gfCNCPoint3[15642] = {X 203.9653, Y 32.4217, Z -4.6667, A 0.000, B 0.000, C 0.000 }
gfCNCPoint3[15643] = {X 206.9865, Y 38.6634, Z -4.6667, A 0.000, B 0.000, C 0.000 }
gfCNCPoint3[15644] = {X 207.4240, Y 39.8017, Z -4.6667, A 0.000, B 0.000, C 0.000 }
gfCNCPoint3[15645] = {X 207.6653, Y 40.9971, Z -4.6667, A 0.000, B 0.000, C 0.000 }
gfCNCPoint3[15646] = {X 207.7038, Y 42.2159, Z -4.6667, A 0.000, B 0.000, C 0.000 }
gfCNCPoint3[15647] = {X 207.5382, Y 43.4241, Z -4.6667, A 0.000, B 0.000, C 0.000 }
gfCNCPoint3[15648] = {X 207.1733, Y 44.5877, Z -4.6667, A 0.000, B 0.000, C 0.000 }
gfCNCPoint3[15649] = {X 206.6193, Y 45.6741, Z -4.6667, A 0.000, B 0.000, C 0.000 }
gfCNCPoint3[15650] = {X 205.8917, Y 46.6527, Z -4.6667, A 0.000, B 0.000, C 0.000 }
gfCNCPoint3[15651] = {X 205.0110, Y 47.4962, Z -4.6667, A 0.000, B 0.000, C 0.000 }
gfCNCPoint3[15652] = {X 204.4743, Y 47.9301, Z -4.6667, A 0.000, B 0.000, C 0.000 }
gfCNCPoint3[15653] = {X 203.5894, Y 48.5431, Z -4.6667, A 0.000, B 0.000, C 0.000 }
gfCNCPoint3[15654] = {X 202.6239, Y 49.0192, Z -4.6667, A 0.000, B 0.000, C 0.000 }
gfCNCPoint3[15655] = {X 201.4894, Y 49.3733, Z -4.6667, A 0.000, B 0.000, C 0.000 }
gfCNCPoint3[15656] = {X 200.3125, Y 49.5385, Z -4.6667, A 0.000, B 0.000, C 0.000 }
gfCNCPoint3[15657] = {X 199.1244, Y 49.5104, Z -4.6667, A 0.000, B 0.000, C 0.000 }
gfCNCPoint3[15658] = {X 196.8334, Y 50.6071, Z -4.6667, A 0.000, B 0.000, C 0.000 }
gfCNCPoint3[15659] = {X 194.4619, Y 51.5166, Z -4.6667, A 0.000, B 0.000, C 0.000 }
gfCNCPoint3[15660] = {X 192.0251, Y 52.2331, Z -4.6667, A 0.000, B 0.000, C 0.000 }
gfCNCPoint3[15661] = {X 190.7222, Y 52.5186, Z -4.6667, A 0.000, B 0.000, C 0.000 }
gfCNCPoint3[15662] = {X 189.4062, Y 52.7359, Z -4.6667, A 0.000, B 0.000, C 0.000 }
gfCNCPoint3[15663] = {X 189.9006, Y 53.9116, Z -4.6667, A 0.000, B 0.000, C 0.000 }
gfCNCPoint3[15664] = {X 190.2683, Y 55.1329, Z -4.6667, A 0.000, B 0.000, C 0.000 }
gfCNCPoint3[15665] = {X 190.5269, Y 56.5561, Z -4.6667, A 0.000, B 0.000, C 0.000 }
gfCNCPoint3[15666] = {X 190.6135, Y 58.0000, Z -4.6667, A 0.000, B 0.000, C 0.000 }
gfCNCPoint3[15667] = {X 190.6132, Y 58.8764, Z -4.6667, A 0.000, B 0.000, C 0.000 }
gfCNCPoint3[15668] = {X 208.6256, Y 78.5346, Z -4.6667, A 0.000, B 0.000, C 0.000 }
gfCNCPoint3[15669] = {X 206.8561, Y 80.1560, Z -4.6667, A 0.000, B 0.000, C 0.000 }
gfCNCPoint3[15670] = {X 213.5228, Y 87.4318, Z -4.6667, A 0.000, B 0.000, C 0.000 }
gfCNCPoint3[15671] = {X 214.2178, Y 87.3794, Z -4.6667, A 0.000, B 0.000, C 0.000 }
gfCNCPoint3[15672] = {X 214.9136, Y 87.3378, Z -4.6667, A 0.000, B 0.000, C 0.000 }
gfCNCPoint3[15673] = {X 234.0915, Y 75.0517, Z -4.6667, A 0.000, B 0.000, C 0.000 }
gfCNCPoint3[15674] = {X 219.6587, Y 69.3879, Z -4.6667, A 0.000, B 0.000, C 0.000 }
gfCNCPoint3[15675] = {X 218.4694, Y 68.9877, Z -4.6667, A 0.000, B 0.000, C 0.000 }
gfCNCPoint3[15676] = {X 217.2420, Y 68.7267, Z -4.6667, A 0.000, B 0.000, C 0.000 }
gfCNCPoint3[15677] = {X 215.9928, Y 68.6082, Z -4.6667, A 0.000, B 0.000, C 0.000 }
gfCNCPoint3[15678] = {X 214.5225, Y 68.4437, Z -4.6667, A 0.000, B 0.000, C 0.000 }
gfCNCPoint3[15679] = {X 213.0946, Y 68.0571, Z -4.6667, A 0.000, B 0.000, C 0.000 }
gfCNCPoint3[15680] = {X 211.7422, Y 67.4574, Z -4.6667, A 0.000, B 0.000, C 0.000 }
gfCNCPoint3[15681] = {X 210.4970, Y 66.6586, Z -4.6667, A 0.000, B 0.000, C 0.000 }
gfCNCPoint3[15682] = {X 209.3880, Y 65.6794, Z -4.6667, A 0.000, B 0.000, C 0.000 }
gfCNCPoint3[15683] = {X 208.4412, Y 64.5427, Z -4.6667, A 0.000, B 0.000, C 0.000 }
gfCNCPoint3[15684] = {X 207.6787, Y 63.2750, Z -4.6667, A 0.000, B 0.000, C 0.000 }
gfCNCPoint3[15685] = {X 207.1183, Y 61.9059, Z -4.6667, A 0.000, B 0.000, C 0.000 }
gfCNCPoint3[15686] = {X 206.7730, Y 60.4673, Z -4.6667, A 0.000, B 0.000, C 0.000 }
gfCNCPoint3[15687] = {X 206.6510, Y 58.9930, Z -4.6667, A 0.000, B 0.000, C 0.000 }
gfCNCPoint3[15688] = {X 206.6508, Y 58.0000, Z -4.6667, A 0.000, B 0.000, C 0.000 }
gfCNCPoint3[15689] = {X 206.7577, Y 56.5655, Z -4.6667, A 0.000, B 0.000, C 0.000 }
gfCNCPoint3[15690] = {X 207.0759, Y 55.1628, Z -4.6667, A 0.000, B 0.000, C 0.000 }
gfCNCPoint3[15691] = {X 207.5986, Y 53.8226, Z -4.6667, A 0.000, B 0.000, C 0.000 }
gfCNCPoint3[15692] = {X 208.3140, Y 52.5747, Z -4.6667, A 0.000, B 0.000, C 0.000 }
gfCNCPoint3[15693] = {X 209.2065, Y 51.4466, Z -4.6667, A 0.000, B 0.000, C 0.000 }
gfCNCPoint3[15694] = {X 210.2563, Y 50.4632, Z -4.6667, A 0.000, B 0.000, C 0.000 }
gfCNCPoint3[15695] = {X 211.4402, Y 49.6463, Z -4.6667, A 0.000, B 0.000, C 0.000 }
gfCNCPoint3[15696] = {X 212.5893, Y 49.0723, Z -4.6667, A 0.000, B 0.000, C 0.000 }
gfCNCPoint3[15697] = {X 213.8042, Y 48.6556, Z -4.6667, A 0.000, B 0.000, C 0.000 }
gfCNCPoint3[15698] = {X 213.2578, Y 48.0874, Z -4.6667, A 0.000, B 0.000, C 0.000 }
gfCNCPoint3[15699] = {X 212.8100, Y 47.4386, Z -4.6667, A 0.000, B 0.000, C 0.000 }
gfCNCPoint3[15700] = {X 212.4725, Y 46.7262, Z -4.6667, A 0.000, B 0.000, C 0.000 }
gfCNCPoint3[15701] = {X 212.2401, Y 45.8965, Z -4.6667, A 0.000, B 0.000, C 0.000 }
gfCNCPoint3[15702] = {X 212.1572, Y 45.0389, Z -4.6667, A 0.000, B 0.000, C 0.000 }
gfCNCPoint3[15703] = {X 212.1570, Y 44.1958, Z -4.6667, A 0.000, B 0.000, C 0.000 }
gfCNCPoint3[15704] = {X 212.2383, Y 43.3151, Z -4.6667, A 0.000, B 0.000, C 0.000 }
gfCNCPoint3[15705] = {X 212.4795, Y 42.4642, Z -4.6667, A 0.000, B 0.000, C 0.000 }
gfCNCPoint3[15706] = {X 212.8723, Y 41.6718, Z -4.6667, A 0.000, B 0.000, C 0.000 }
gfCNCPoint3[15707] = {X 213.4036, Y 40.9647, Z -4.6667, A 0.000, B 0.000, C 0.000 }
gfCNCPoint3[15708] = {X 213.6821, Y 40.6575, Z -4.6667, A 0.000, B 0.000, C 0.000 }
gfCNCPoint3[15709] = {X 213.6849, Y 40.3041, Z -4.6667, A 0.000, B 0.000, C 0.000 }
gfCNCPoint3[15710] = {X 213.6849, Y 17.4645, Z -4.6667, A 0.000, B 0.000, C 0.000 }
gfCNCPoint3[15711] = {X 213.6795, Y 16.7696, Z -4.6667, A 0.000, B 0.000, C 0.000 }
gfCNCPoint3[15712] = {X 213.6793, Y 16.5192, Z -4.6667, A 0.000, B 0.000, C 0.000 }
gfCNCPoint3[15713] = {X 213.0402, Y 15.7779, Z -4.6667, A 0.000, B 0.000, C 0.000 }
gfCNCPoint3[15714] = {X 212.5618, Y 14.9240, Z -4.6667, A 0.000, B 0.000, C 0.000 }
gfCNCPoint3[15715] = {X 212.2635, Y 13.9918, Z -4.6667, A 0.000, B 0.000, C 0.000 }
gfCNCPoint3[15716] = {X 212.1572, Y 13.0188, Z -4.6667, A 0.000, B 0.000, C 0.000 }
gfCNCPoint3[15717] = {X 212.1570, Y 12.1868, Z -4.6667, A 0.000, B 0.000, C 0.000 }
gfCNCPoint3[15718] = {X 212.2436, Y 11.2717, Z -4.6667, A 0.000, B 0.000, C 0.000 }
gfCNCPoint3[15719] = {X 212.5002, Y 10.3891, Z -4.6667, A 0.000, B 0.000, C 0.000 }
gfCNCPoint3[15720] = {X 212.9449, Y 9.5280, Z -4.6667, A 0.000, B 0.000, C 0.000 }
gfCNCPoint3[15721] = {X 213.5510, Y 8.7718, Z -4.6667, A 0.000, B 0.000, C 0.000 }
gfCNCPoint3[15722] = {X 214.2946, Y 8.1503, Z -4.6667, A 0.000, B 0.000, C 0.000 }
gfCNCPoint3[15723] = {X 215.1464, Y 7.6879, Z -4.6667, A 0.000, B 0.000, C 0.000 }
gfCNCPoint3[15724] = {X 216.0727, Y 7.4030, Z -4.6667, A 0.000, B 0.000, C 0.000 }
gfCNCPoint3[15725] = {X 217.0370, Y 7.3068, Z -4.6667, A 0.000, B 0.000, C 0.000 }
gfCNCPoint3[15726] = {X 223.4805, Y 7.3068, Z -4.6667, A 0.000, B 0.000, C 0.000 }
gfCNCPoint3[15727] = {X 224.4448, Y 7.4030, Z -4.6667, A 0.000, B 0.000, C 0.000 }
gfCNCPoint3[15728] = {X 225.3711, Y 7.6879, Z -4.6667, A 0.000, B 0.000, C 0.000 }
gfCNCPoint3[15729] = {X 226.2229, Y 8.1503, Z -4.6667, A 0.000, B 0.000, C 0.000 }
gfCNCPoint3[15730] = {X 226.9665, Y 8.7718, Z -4.6667, A 0.000, B 0.000, C 0.000 }
gfCNCPoint3[15731] = {X 227.5726, Y 9.5280, Z -4.6667, A 0.000, B 0.000, C 0.000 }
gfCNCPoint3[15732] = {X 228.0173, Y 10.3891, Z -4.6667, A 0.000, B 0.000, C 0.000 }
gfCNCPoint3[15733] = {X 228.2739, Y 11.2717, Z -4.6667, A 0.000, B 0.000, C 0.000 }
gfCNCPoint3[15734] = {X 228.3605, Y 12.1868, Z -4.6667, A 0.000, B 0.000, C 0.000 }
gfCNCPoint3[15735] = {X 228.3603, Y 13.0237, Z -4.6667, A 0.000, B 0.000, C 0.000 }
gfCNCPoint3[15736] = {X 228.2529, Y 13.9971, Z -4.6667, A 0.000, B 0.000, C 0.000 }
gfCNCPoint3[15737] = {X 227.9533, Y 14.9294, Z -4.6667, A 0.000, B 0.000, C 0.000 }
gfCNCPoint3[15738] = {X 227.4737, Y 15.7831, Z -4.6667, A 0.000, B 0.000, C 0.000 }
gfCNCPoint3[15739] = {X 226.8333, Y 16.5239, Z -4.6667, A 0.000, B 0.000, C 0.000 }
gfCNCPoint3[15740] = {X 226.8342, Y 40.6638, Z -4.6667, A 0.000, B 0.000, C 0.000 }
gfCNCPoint3[15741] = {X 227.4743, Y 41.4046, Z -4.6667, A 0.000, B 0.000, C 0.000 }
gfCNCPoint3[15742] = {X 227.9537, Y 42.2583, Z -4.6667, A 0.000, B 0.000, C 0.000 }
gfCNCPoint3[15743] = {X 228.2531, Y 43.1906, Z -4.6667, A 0.000, B 0.000, C 0.000 }
gfCNCPoint3[15744] = {X 228.3603, Y 44.1638, Z -4.6667, A 0.000, B 0.000, C 0.000 }
gfCNCPoint3[15745] = {X 228.3605, Y 45.0000, Z -4.6667, A 0.000, B 0.000, C 0.000 }
gfCNCPoint3[15746] = {X 228.3507, Y 45.3090, Z -4.6667, A 0.000, B 0.000, C 0.000 }
gfCNCPoint3[15747] = {X 228.3214, Y 45.6167, Z -4.6667, A 0.000, B 0.000, C 0.000 }
gfCNCPoint3[15748] = {X 228.0910, Y 46.5992, Z -4.6667, A 0.000, B 0.000, C 0.000 }
gfCNCPoint3[15749] = {X 227.6635, Y 47.5134, Z -4.6667, A 0.000, B 0.000, C 0.000 }
gfCNCPoint3[15750] = {X 227.0571, Y 48.3200, Z -4.6667, A 0.000, B 0.000, C 0.000 }
gfCNCPoint3[15751] = {X 226.7053, Y 47.9934, Z -4.6667, A 0.000, B 0.000, C 0.000 }
gfCNCPoint3[15752] = {X 226.0261, Y 48.5889, Z -4.6667, A 0.000, B 0.000, C 0.000 }
gfCNCPoint3[15753] = {X 225.2396, Y 49.0331, Z -4.6667, A 0.000, B 0.000, C 0.000 }
gfCNCPoint3[15754] = {X 224.3790, Y 49.3073, Z -4.6667, A 0.000, B 0.000, C 0.000 }
gfCNCPoint3[15755] = {X 223.4805, Y 49.4000, Z -4.6667, A 0.000, B 0.000, C 0.000 }
gfCNCPoint3[15756] = {X 217.0370, Y 49.4000, Z -4.6667, A 0.000, B 0.000, C 0.000 }
gfCNCPoint3[15757] = {X 216.0579, Y 49.2897, Z -4.6667, A 0.000, B 0.000, C 0.000 }
gfCNCPoint3[15758] = {X 215.1279, Y 48.9643, Z -4.6667, A 0.000, B 0.000, C 0.000 }
gfCNCPoint3[15759] = {X 214.2936, Y 48.4400, Z -4.6667, A 0.000, B 0.000, C 0.000 }
gfCNCPoint3[15760] = {X 213.5969, Y 47.7433, Z -4.6667, A 0.000, B 0.000, C 0.000 }
gfCNCPoint3[15761] = {X 213.0727, Y 46.9091, Z -4.6667, A 0.000, B 0.000, C 0.000 }
gfCNCPoint3[15762] = {X 212.7473, Y 45.9791, Z -4.6667, A 0.000, B 0.000, C 0.000 }
gfCNCPoint3[15763] = {X 212.6370, Y 45.0000, Z -4.6667, A 0.000, B 0.000, C 0.000 }
gfCNCPoint3[15764] = {X 212.6370, Y 44.1958, Z -4.6667, A 0.000, B 0.000, C 0.000 }
gfCNCPoint3[15765] = {X 212.7102, Y 43.4029, Z -4.6667, A 0.000, B 0.000, C 0.000 }
gfCNCPoint3[15766] = {X 212.9273, Y 42.6369, Z -4.6667, A 0.000, B 0.000, C 0.000 }
gfCNCPoint3[15767] = {X 213.2810, Y 41.9236, Z -4.6667, A 0.000, B 0.000, C 0.000 }
gfCNCPoint3[15768] = {X 213.7592, Y 41.2871, Z -4.6667, A 0.000, B 0.000, C 0.000 }
gfCNCPoint3[15769] = {X 214.1607, Y 40.8442, Z -4.6667, A 0.000, B 0.000, C 0.000 }
gfCNCPoint3[15770] = {X 214.1649, Y 40.3060, Z -4.6667, A 0.000, B 0.000, C 0.000 }
gfCNCPoint3[15771] = {X 214.1649, Y 17.4626, Z -4.6667, A 0.000, B 0.000, C 0.000 }
gfCNCPoint3[15772] = {X 214.1595, Y 16.7692, Z -4.6667, A 0.000, B 0.000, C 0.000 }
gfCNCPoint3[15773] = {X 214.1591, Y 16.3063, Z -4.6667, A 0.000, B 0.000, C 0.000 }
gfCNCPoint3[15774] = {X 213.5167, Y 15.6176, Z -4.6667, A 0.000, B 0.000, C 0.000 }
gfCNCPoint3[15775] = {X 213.0356, Y 14.8079, Z -4.6667, A 0.000, B 0.000, C 0.000 }
gfCNCPoint3[15776] = {X 212.7378, Y 13.9144, Z -4.6667, A 0.000, B 0.000, C 0.000 }
gfCNCPoint3[15777] = {X 212.6370, Y 12.9779, Z -4.6667, A 0.000, B 0.000, C 0.000 }
gfCNCPoint3[15778] = {X 212.6370, Y 12.1868, Z -4.6667, A 0.000, B 0.000, C 0.000 }
gfCNCPoint3[15779] = {X 212.7473, Y 11.2077, Z -4.6667, A 0.000, B 0.000, C 0.000 }
gfCNCPoint3[15780] = {X 213.0728, Y 10.2777, Z -4.6667, A 0.000, B 0.000, C 0.000 }
gfCNCPoint3[15781] = {X 213.5970, Y 9.4435, Z -4.6667, A 0.000, B 0.000, C 0.000 }
gfCNCPoint3[15782] = {X 214.2937, Y 8.7468, Z -4.6667, A 0.000, B 0.000, C 0.000 }
gfCNCPoint3[15783] = {X 215.1279, Y 8.2226, Z -4.6667, A 0.000, B 0.000, C 0.000 }
gfCNCPoint3[15784] = {X 216.0579, Y 7.8971, Z -4.6667, A 0.000, B 0.000, C 0.000 }
gfCNCPoint3[15785] = {X 217.0370, Y 7.7868, Z -4.6667, A 0.000, B 0.000, C 0.000 }
gfCNCPoint3[15786] = {X 223.4805, Y 7.7868, Z -4.6667, A 0.000, B 0.000, C 0.000 }
gfCNCPoint3[15787] = {X 224.4596, Y 7.8971, Z -4.6667, A 0.000, B 0.000, C 0.000 }
gfCNCPoint3[15788] = {X 225.3896, Y 8.2226, Z -4.6667, A 0.000, B 0.000, C 0.000 }
gfCNCPoint3[15789] = {X 226.2238, Y 8.7468, Z -4.6667, A 0.000, B 0.000, C 0.000 }
gfCNCPoint3[15790] = {X 226.9205, Y 9.4435, Z -4.6667, A 0.000, B 0.000, C 0.000 }
gfCNCPoint3[15791] = {X 227.4447, Y 10.2777, Z -4.6667, A 0.000, B 0.000, C 0.000 }
gfCNCPoint3[15792] = {X 227.7702, Y 11.2077, Z -4.6667, A 0.000, B 0.000, C 0.000 }
gfCNCPoint3[15793] = {X 227.8805, Y 12.1868, Z -4.6667, A 0.000, B 0.000, C 0.000 }
gfCNCPoint3[15794] = {X 227.8802, Y 13.0233, Z -4.6667, A 0.000, B 0.000, C 0.000 }
gfCNCPoint3[15795] = {X 227.7720, Y 13.9493, Z -4.6667, A 0.000, B 0.000, C 0.000 }
gfCNCPoint3[15796] = {X 227.4710, Y 14.8316, Z -4.6667, A 0.000, B 0.000, C 0.000 }
gfCNCPoint3[15797] = {X 226.9909, Y 15.6307, Z -4.6667, A 0.000, B 0.000, C 0.000 }
gfCNCPoint3[15798] = {X 226.3532, Y 16.3108, Z -4.6667, A 0.000, B 0.000, C 0.000 }
gfCNCPoint3[15799] = {X 226.3542, Y 40.8768, Z -4.6667, A 0.000, B 0.000, C 0.000 }
gfCNCPoint3[15800] = {X 226.9983, Y 41.5659, Z -4.6667, A 0.000, B 0.000, C 0.000 }
gfCNCPoint3[15801] = {X 227.4808, Y 42.3764, Z -4.6667, A 0.000, B 0.000, C 0.000 }
gfCNCPoint3[15802] = {X 227.7794, Y 43.2711, Z -4.6667, A 0.000, B 0.000, C 0.000 }
gfCNCPoint3[15803] = {X 227.8805, Y 44.2089, Z -4.6667, A 0.000, B 0.000, C 0.000 }
gfCNCPoint3[15804] = {X 227.8805, Y 45.0000, Z -4.6667, A 0.000, B 0.000, C 0.000 }
gfCNCPoint3[15805] = {X 227.8037, Y 45.8182, Z -4.6667, A 0.000, B 0.000, C 0.000 }
gfCNCPoint3[15806] = {X 227.5762, Y 46.6079, Z -4.6667, A 0.000, B 0.000, C 0.000 }
gfCNCPoint3[15807] = {X 227.2057, Y 47.3415, Z -4.6667, A 0.000, B 0.000, C 0.000 }
gfCNCPoint3[15808] = {X 226.7053, Y 47.9934, Z -4.6667, A 0.000, B 0.000, C 0.000 }
gfCNCPoint3[15809] = {X 227.0571, Y 48.3200, Z -4.6667, A 0.000, B 0.000, C 0.000 }
gfCNCPoint3[15810] = {X 236.2309, Y 48.3200, Z -4.6667, A 0.000, B 0.000, C 0.000 }
gfCNCPoint3[15811] = {X 235.6245, Y 47.5134, Z -4.6667, A 0.000, B 0.000, C 0.000 }
gfCNCPoint3[15812] = {X 235.1970, Y 46.5992, Z -4.6667, A 0.000, B 0.000, C 0.000 }
gfCNCPoint3[15813] = {X 234.9666, Y 45.6167, Z -4.6667, A 0.000, B 0.000, C 0.000 }
gfCNCPoint3[15814] = {X 234.9373, Y 45.3090, Z -4.6667, A 0.000, B 0.000, C 0.000 }
gfCNCPoint3[15815] = {X 234.9275, Y 45.0000, Z -4.6667, A 0.000, B 0.000, C 0.000 }
gfCNCPoint3[15816] = {X 234.9275, Y 44.2089, Z -4.6667, A 0.000, B 0.000, C 0.000 }
gfCNCPoint3[15817] = {X 235.0194, Y 43.2661, Z -4.6667, A 0.000, B 0.000, C 0.000 }
gfCNCPoint3[15818] = {X 235.2917, Y 42.3588, Z -4.6667, A 0.000, B 0.000, C 0.000 }
gfCNCPoint3[15819] = {X 235.7342, Y 41.5212, Z -4.6667, A 0.000, B 0.000, C 0.000 }
gfCNCPoint3[15820] = {X 236.3302, Y 40.7849, Z -4.6667, A 0.000, B 0.000, C 0.000 }
gfCNCPoint3[15821] = {X 237.0572, Y 40.1776, Z -4.6667, A 0.000, B 0.000, C 0.000 }
gfCNCPoint3[15822] = {X 237.8878, Y 39.7222, Z -4.6667, A 0.000, B 0.000, C 0.000 }
gfCNCPoint3[15823] = {X 241.5463, Y 32.5611, Z -4.6667, A 0.000, B 0.000, C 0.000 }
gfCNCPoint3[15824] = {X 240.2118, Y 31.5584, Z -4.6667, A 0.000, B 0.000, C 0.000 }
gfCNCPoint3[15825] = {X 239.0310, Y 30.3785, Z -4.6667, A 0.000, B 0.000, C 0.000 }
gfCNCPoint3[15826] = {X 238.0273, Y 29.0447, Z -4.6667, A 0.000, B 0.000, C 0.000 }
gfCNCPoint3[15827] = {X 237.2205, Y 27.5834, Z -4.6667, A 0.000, B 0.000, C 0.000 }
gfCNCPoint3[15828] = {X 236.6265, Y 26.0235, Z -4.6667, A 0.000, B 0.000, C 0.000 }
gfCNCPoint3[15829] = {X 236.1914, Y 24.1499, Z -4.6667, A 0.000, B 0.000, C 0.000 }
gfCNCPoint3[15830] = {X 235.9695, Y 22.2393, Z -4.6667, A 0.000, B 0.000, C 0.000 }
gfCNCPoint3[15831] = {X 235.9636, Y 20.3158, Z -4.6667, A 0.000, B 0.000, C 0.000 }
gfCNCPoint3[15832] = {X 236.1739, Y 18.4039, Z -4.6667, A 0.000, B 0.000, C 0.000 }
gfCNCPoint3[15833] = {X 236.5975, Y 16.5277, Z -4.6667, A 0.000, B 0.000, C 0.000 }
gfCNCPoint3[15834] = {X 237.1169, Y 15.0571, Z -4.6667, A 0.000, B 0.000, C 0.000 }
gfCNCPoint3[15835] = {X 237.8166, Y 13.6632, Z -4.6667, A 0.000, B 0.000, C 0.000 }
gfCNCPoint3[15836] = {X 238.6856, Y 12.3681, Z -4.6667, A 0.000, B 0.000, C 0.000 }
gfCNCPoint3[15837] = {X 239.7103, Y 11.1923, Z -4.6667, A 0.000, B 0.000, C 0.000 }
gfCNCPoint3[15838] = {X 240.8746, Y 10.1541, Z -4.6667, A 0.000, B 0.000, C 0.000 }
gfCNCPoint3[15839] = {X 242.1599, Y 9.2702, Z -4.6667, A 0.000, B 0.000, C 0.000 }
gfCNCPoint3[15840] = {X 243.5460, Y 8.5546, Z -4.6667, A 0.000, B 0.000, C 0.000 }
gfCNCPoint3[15841] = {X 245.0110, Y 8.0185, Z -4.6667, A 0.000, B 0.000, C 0.000 }
gfCNCPoint3[15842] = {X 246.5316, Y 7.6705, Z -4.6667, A 0.000, B 0.000, C 0.000 }
gfCNCPoint3[15843] = {X 248.6761, Y 7.3930, Z -4.6667, A 0.000, B 0.000, C 0.000 }
gfCNCPoint3[15844] = {X 250.8369, Y 7.3106, Z -4.6667, A 0.000, B 0.000, C 0.000 }
gfCNCPoint3[15845] = {X 266.7608, Y 7.3106, Z -4.6667, A 0.000, B 0.000, C 0.000 }
gfCNCPoint3[15846] = {X 267.7191, Y 7.4120, Z -4.6667, A 0.000, B 0.000, C 0.000 }
gfCNCPoint3[15847] = {X 268.6388, Y 7.6997, Z -4.6667, A 0.000, B 0.000, C 0.000 }
gfCNCPoint3[15848] = {X 269.4841, Y 8.1624, Z -4.6667, A 0.000, B 0.000, C 0.000 }
gfCNCPoint3[15849] = {X 270.2221, Y 8.7821, Z -4.6667, A 0.000, B 0.000, C 0.000 }
gfCNCPoint3[15850] = {X 270.8239, Y 9.5347, Z -4.6667, A 0.000, B 0.000, C 0.000 }
gfCNCPoint3[15851] = {X 271.2663, Y 10.3908, Z -4.6667, A 0.000, B 0.000, C 0.000 }
gfCNCPoint3[15852] = {X 271.5234, Y 11.2719, Z -4.6667, A 0.000, B 0.000, C 0.000 }
gfCNCPoint3[15853] = {X 271.6110, Y 12.1855, Z -4.6667, A 0.000, B 0.000, C 0.000 }
gfCNCPoint3[15854] = {X 271.6108, Y 13.0237, Z -4.6667, A 0.000, B 0.000, C 0.000 }
gfCNCPoint3[15855] = {X 271.5128, Y 13.9524, Z -4.6667, A 0.000, B 0.000, C 0.000 }
gfCNCPoint3[15856] = {X 271.2396, Y 14.8453, Z -4.6667, A 0.000, B 0.000, C 0.000 }
gfCNCPoint3[15857] = {X 275.6743, Y 16.6820, Z -4.6667, A 0.000, B 0.000, C 0.000 }
gfCNCPoint3[15858] = {X 275.3127, Y 17.4566, Z -4.6667, A 0.000, B 0.000, C 0.000 }
gfCNCPoint3[15859] = {X 274.8840, Y 18.1964, Z -4.6667, A 0.000, B 0.000, C 0.000 }
gfCNCPoint3[15860] = {X 274.8839, Y 38.9902, Z -4.6667, A 0.000, B 0.000, C 0.000 }
gfCNCPoint3[15861] = {X 275.3140, Y 39.7327, Z -4.6667, A 0.000, B 0.000, C 0.000 }
gfCNCPoint3[15862] = {X 275.6766, Y 40.5104, Z -4.6667, A 0.000, B 0.000, C 0.000 }
gfCNCPoint3[15863] = {X 276.0377, Y 39.7359, Z -4.6667, A 0.000, B 0.000, C 0.000 }
gfCNCPoint3[15864] = {X 276.4653, Y 38.9961, Z -4.6667, A 0.000, B 0.000, C 0.000 }
gfCNCPoint3[15865] = {X 276.4649, Y 18.1968, Z -4.6667, A 0.000, B 0.000, C 0.000 }
gfCNCPoint3[15866] = {X 276.0362, Y 17.4569, Z -4.6667, A 0.000, B 0.000, C 0.000 }
gfCNCPoint3[15867] = {X 275.6743, Y 16.6820, Z -4.6667, A 0.000, B 0.000, C 0.000 }
gfCNCPoint3[15868] = {X 273.4570, Y 15.7637, Z -4.6667, A 0.000, B 0.000, C 0.000 }
gfCNCPoint3[15869] = {X 273.0265, Y 16.6339, Z -4.6667, A 0.000, B 0.000, C 0.000 }
gfCNCPoint3[15870] = {X 272.4840, Y 17.4391, Z -4.6667, A 0.000, B 0.000, C 0.000 }
gfCNCPoint3[15871] = {X 272.4839, Y 39.7475, Z -4.6667, A 0.000, B 0.000, C 0.000 }
gfCNCPoint3[15872] = {X 273.0276, Y 40.5547, Z -4.6667, A 0.000, B 0.000, C 0.000 }
gfCNCPoint3[15873] = {X 273.4587, Y 41.4273, Z -4.6667, A 0.000, B 0.000, C 0.000 }
gfCNCPoint3[15874] = {X 273.7589, Y 42.3094, Z -4.6667, A 0.000, B 0.000, C 0.000 }
gfCNCPoint3[15875] = {X 273.9439, Y 43.2225, Z -4.6667, A 0.000, B 0.000, C 0.000 }
gfCNCPoint3[15876] = {X 274.0108, Y 44.1519, Z -4.6667, A 0.000, B 0.000, C 0.000 }
gfCNCPoint3[15877] = {X 274.0110, Y 45.0000, Z -4.6667, A 0.000, B 0.000, C 0.000 }
gfCNCPoint3[15878] = {X 273.9884, Y 45.5734, Z -4.6667, A 0.000, B 0.000, C 0.000 }
gfCNCPoint3[15879] = {X 273.9207, Y 46.1433, Z -4.6667, A 0.000, B 0.000, C 0.000 }
gfCNCPoint3[15880] = {X 275.0713, Y 45.9760, Z -4.6667, A 0.000, B 0.000, C 0.000 }
gfCNCPoint3[15881] = {X 276.2327, Y 45.9200, Z -4.6667, A 0.000, B 0.000, C 0.000 }
gfCNCPoint3[15882] = {X 277.3960, Y 45.9200, Z -4.6667, A 0.000, B 0.000, C 0.000 }
gfCNCPoint3[15883] = {X 277.3539, Y 45.4857, Z -4.6667, A 0.000, B 0.000, C 0.000 }
gfCNCPoint3[15884] = {X 277.3378, Y 45.0498, Z -4.6667, A 0.000, B 0.000, C 0.000 }
gfCNCPoint3[15885] = {X 277.3377, Y 44.1984, Z -4.6667, A 0.000, B 0.000, C 0.000 }
gfCNCPoint3[15886] = {X 277.4029, Y 43.2534, Z -4.6667, A 0.000, B 0.000, C 0.000 }
gfCNCPoint3[15887] = {X 277.5895, Y 42.3247, Z -4.6667, A 0.000, B 0.000, C 0.000 }
gfCNCPoint3[15888] = {X 277.8943, Y 41.4279, Z -4.6667, A 0.000, B 0.000, C 0.000 }
gfCNCPoint3[15889] = {X 278.3242, Y 40.5572, Z -4.6667, A 0.000, B 0.000, C 0.000 }
gfCNCPoint3[15890] = {X 278.8653, Y 39.7510, Z -4.6667, A 0.000, B 0.000, C 0.000 }
gfCNCPoint3[15891] = {X 278.8649, Y 17.4394, Z -4.6667, A 0.000, B 0.000, C 0.000 }
gfCNCPoint3[15892] = {X 278.3223, Y 16.6341, Z -4.6667, A 0.000, B 0.000, C 0.000 }
gfCNCPoint3[15893] = {X 277.8917, Y 15.7637, Z -4.6667, A 0.000, B 0.000, C 0.000 }
gfCNCPoint3[15894] = {X 277.5902, Y 14.8788, Z -4.6667, A 0.000, B 0.000, C 0.000 }
gfCNCPoint3[15895] = {X 277.4046, Y 13.9627, Z -4.6667, A 0.000, B 0.000, C 0.000 }
gfCNCPoint3[15896] = {X 277.3379, Y 13.0303, Z -4.6667, A 0.000, B 0.000, C 0.000 }
gfCNCPoint3[15897] = {X 277.3377, Y 12.1868, Z -4.6667, A 0.000, B 0.000, C 0.000 }
gfCNCPoint3[15898] = {X 277.3952, Y 11.2737, Z -4.6667, A 0.000, B 0.000, C 0.000 }
gfCNCPoint3[15899] = {X 277.5667, Y 10.3750, Z -4.6667, A 0.000, B 0.000, C 0.000 }
gfCNCPoint3[15900] = {X 277.8496, Y 9.5050, Z -4.6667, A 0.000, B 0.000, C 0.000 }
gfCNCPoint3[15901] = {X 273.4968, Y 9.5050, Z -4.6667, A 0.000, B 0.000, C 0.000 }
gfCNCPoint3[15902] = {X 273.7800, Y 10.3733, Z -4.6667, A 0.000, B 0.000, C 0.000 }
gfCNCPoint3[15903] = {X 273.9524, Y 11.2703, Z -4.6667, A 0.000, B 0.000, C 0.000 }
gfCNCPoint3[15904] = {X 274.0110, Y 12.1819, Z -4.6667, A 0.000, B 0.000, C 0.000 }
gfCNCPoint3[15905] = {X 274.0107, Y 13.0462, Z -4.6667, A 0.000, B 0.000, C 0.000 }
gfCNCPoint3[15906] = {X 273.9427, Y 13.9732, Z -4.6667, A 0.000, B 0.000, C 0.000 }
gfCNCPoint3[15907] = {X 273.7571, Y 14.8840, Z -4.6667, A 0.000, B 0.000, C 0.000 }
gfCNCPoint3[15908] = {X 273.4570, Y 15.7637, Z -4.6667, A 0.000, B 0.000, C 0.000 }
gfCNCPoint3[15909] = {X 271.2396, Y 14.8453, Z -4.6667, A 0.000, B 0.000, C 0.000 }
gfCNCPoint3[15910] = {X 270.7504, Y 15.7455, Z -4.6667, A 0.000, B 0.000, C 0.000 }
gfCNCPoint3[15911] = {X 270.0840, Y 16.5237, Z -4.6667, A 0.000, B 0.000, C 0.000 }
gfCNCPoint3[15912] = {X 270.0839, Y 40.6630, Z -4.6667, A 0.000, B 0.000, C 0.000 }
gfCNCPoint3[15913] = {X 270.7243, Y 41.4038, Z -4.6667, A 0.000, B 0.000, C 0.000 }
gfCNCPoint3[15914] = {X 271.2040, Y 42.2576, Z -4.6667, A 0.000, B 0.000, C 0.000 }
gfCNCPoint3[15915] = {X 271.5035, Y 43.1899, Z -4.6667, A 0.000, B 0.000, C 0.000 }
gfCNCPoint3[15916] = {X 271.6108, Y 44.1633, Z -4.6667, A 0.000, B 0.000, C 0.000 }
gfCNCPoint3[15917] = {X 271.6110, Y 45.0000, Z -4.6667, A 0.000, B 0.000, C 0.000 }
gfCNCPoint3[15918] = {X 271.5959, Y 45.3844, Z -4.6667, A 0.000, B 0.000, C 0.000 }
gfCNCPoint3[15919] = {X 271.5505, Y 45.7664, Z -4.6667, A 0.000, B 0.000, C 0.000 }
gfCNCPoint3[15920] = {X 271.2989, Y 46.7171, Z -4.6667, A 0.000, B 0.000, C 0.000 }
gfCNCPoint3[15921] = {X 270.8619, Y 47.5982, Z -4.6667, A 0.000, B 0.000, C 0.000 }
gfCNCPoint3[15922] = {X 270.2571, Y 48.3736, Z -4.6667, A 0.000, B 0.000, C 0.000 }
gfCNCPoint3[15923] = {X 269.5090, Y 49.0121, Z -4.6667, A 0.000, B 0.000, C 0.000 }
gfCNCPoint3[15924] = {X 268.6482, Y 49.4876, Z -4.6667, A 0.000, B 0.000, C 0.000 }
gfCNCPoint3[15925] = {X 267.7095, Y 49.7809, Z -4.6667, A 0.000, B 0.000, C 0.000 }
gfCNCPoint3[15926] = {X 266.7310, Y 49.8800, Z -4.6667, A 0.000, B 0.000, C 0.000 }
gfCNCPoint3[15927] = {X 262.1384, Y 49.8800, Z -4.6667, A 0.000, B 0.000, C 0.000 }
gfCNCPoint3[15928] = {X 262.1384, Y 54.6800, Z -4.6667, A 0.000, B 0.000, C 0.000 }
gfCNCPoint3[15929] = {X 260.2870, Y 54.6800, Z -4.6667, A 0.000, B 0.000, C 0.000 }
gfCNCPoint3[15930] = {X 261.9957, Y 55.3582, Z -4.6667, A 0.000, B 0.000, C 0.000 }
gfCNCPoint3[15931] = {X 262.0630, Y 55.0183, Z -4.6667, A 0.000, B 0.000, C 0.000 }
gfCNCPoint3[15932] = {X 262.1384, Y 54.6800, Z -4.6667, A 0.000, B 0.000, C 0.000 }
gfCNCPoint3[15933] = {X 262.1384, Y 52.2800, Z -4.6667, A 0.000, B 0.000, C 0.000 }
gfCNCPoint3[15934] = {X 260.2876, Y 52.2800, Z -4.6667, A 0.000, B 0.000, C 0.000 }
gfCNCPoint3[15935] = {X 259.1915, Y 52.1970, Z -4.6667, A 0.000, B 0.000, C 0.000 }
gfCNCPoint3[15936] = {X 258.1205, Y 51.9500, Z -4.6667, A 0.000, B 0.000, C 0.000 }
gfCNCPoint3[15937] = {X 257.0989, Y 51.5445, Z -4.6667, A 0.000, B 0.000, C 0.000 }
gfCNCPoint3[15938] = {X 256.1499, Y 50.9898, Z -4.6667, A 0.000, B 0.000, C 0.000 }
gfCNCPoint3[15939] = {X 255.2953, Y 50.2986, Z -4.6667, A 0.000, B 0.000, C 0.000 }
gfCNCPoint3[15940] = {X 253.6495, Y 52.0454, Z -4.6667, A 0.000, B 0.000, C 0.000 }
gfCNCPoint3[15941] = {X 253.4933, Y 51.8950, Z -4.6667, A 0.000, B 0.000, C 0.000 }
gfCNCPoint3[15942] = {X 253.3406, Y 51.7410, Z -4.6667, A 0.000, B 0.000, C 0.000 }
gfCNCPoint3[15943] = {X 253.2763, Y 51.8066, Z -4.6667, A 0.000, B 0.000, C 0.000 }
gfCNCPoint3[15944] = {X 253.2115, Y 51.8716, Z -4.6667, A 0.000, B 0.000, C 0.000 }
gfCNCPoint3[15945] = {X 253.6495, Y 52.0454, Z -4.6667, A 0.000, B 0.000, C 0.000 }
gfCNCPoint3[15946] = {X 255.2953, Y 50.2986, Z -4.6667, A 0.000, B 0.000, C 0.000 }
gfCNCPoint3[15947] = {X 255.1778, Y 50.1855, Z -4.6667, A 0.000, B 0.000, C 0.000 }
gfCNCPoint3[15948] = {X 255.0630, Y 50.0697, Z -4.6667, A 0.000, B 0.000, C 0.000 }
gfCNCPoint3[15949] = {X 254.3405, Y 49.1989, Z -4.6667, A 0.000, B 0.000, C 0.000 }
gfCNCPoint3[15950] = {X 253.7617, Y 48.2267, Z -4.6667, A 0.000, B 0.000, C 0.000 }
gfCNCPoint3[15951] = {X 253.3406, Y 47.1766, Z -4.6667, A 0.000, B 0.000, C 0.000 }
gfCNCPoint3[15952] = {X 252.9194, Y 48.2267, Z -4.6667, A 0.000, B 0.000, C 0.000 }
gfCNCPoint3[15953] = {X 252.3406, Y 49.1989, Z -4.6667, A 0.000, B 0.000, C 0.000 }
gfCNCPoint3[15954] = {X 251.6182, Y 50.0697, Z -4.6667, A 0.000, B 0.000, C 0.000 }
gfCNCPoint3[15955] = {X 251.5699, Y 50.1190, Z -4.6667, A 0.000, B 0.000, C 0.000 }
gfCNCPoint3[15956] = {X 251.5211, Y 50.1679, Z -4.6667, A 0.000, B 0.000, C 0.000 }
gfCNCPoint3[15957] = {X 250.7151, Y 50.8585, Z -4.6667, A 0.000, B 0.000, C 0.000 }
gfCNCPoint3[15958] = {X 249.8174, Y 51.4246, Z -4.6667, A 0.000, B 0.000, C 0.000 }
gfCNCPoint3[15959] = {X 248.8468, Y 51.8542, Z -4.6667, A 0.000, B 0.000, C 0.000 }
gfCNCPoint3[15960] = {X 247.8241, Y 52.1381, Z -4.6667, A 0.000, B 0.000, C 0.000 }
gfCNCPoint3[15961] = {X 247.8929, Y 52.2638, Z -4.6667, A 0.000, B 0.000, C 0.000 }
gfCNCPoint3[15962] = {X 247.9602, Y 52.3904, Z -4.6667, A 0.000, B 0.000, C 0.000 }
gfCNCPoint3[15963] = {X 250.9674, Y 53.5630, Z -4.6667, A 0.000, B 0.000, C 0.000 }
gfCNCPoint3[15964] = {X 264.1528, Y 58.7966, Z -4.6667, A 0.000, B 0.000, C 0.000 }
gfCNCPoint3[15965] = {X 264.1527, Y 58.0000, Z -4.6667, A 0.000, B 0.000, C 0.000 }
gfCNCPoint3[15966] = {X 264.2035, Y 56.8934, Z -4.6667, A 0.000, B 0.000, C 0.000 }
gfCNCPoint3[15967] = {X 264.3554, Y 55.7961, Z -4.6667, A 0.000, B 0.000, C 0.000 }
gfCNCPoint3[15968] = {X 264.4116, Y 55.5125, Z -4.6667, A 0.000, B 0.000, C 0.000 }
gfCNCPoint3[15969] = {X 264.4745, Y 55.2303, Z -4.6667, A 0.000, B 0.000, C 0.000 }
gfCNCPoint3[15970] = {X 264.9369, Y 53.7185, Z -4.6667, A 0.000, B 0.000, C 0.000 }
gfCNCPoint3[15971] = {X 265.5928, Y 52.2800, Z -4.6667, A 0.000, B 0.000, C 0.000 }
gfCNCPoint3[15972] = {X 262.1384, Y 52.2800, Z -4.6667, A 0.000, B 0.000, C 0.000 }
gfCNCPoint3[15973] = {X 262.1384, Y 49.8800, Z -4.6667, A 0.000, B 0.000, C 0.000 }
gfCNCPoint3[15974] = {X 260.2876, Y 49.8800, Z -4.6667, A 0.000, B 0.000, C 0.000 }
gfCNCPoint3[15975] = {X 259.2646, Y 49.7716, Z -4.6667, A 0.000, B 0.000, C 0.000 }
gfCNCPoint3[15976] = {X 258.2870, Y 49.4511, Z -4.6667, A 0.000, B 0.000, C 0.000 }
gfCNCPoint3[15977] = {X 257.3984, Y 48.9328, Z -4.6667, A 0.000, B 0.000, C 0.000 }
gfCNCPoint3[15978] = {X 256.6382, Y 48.2398, Z -4.6667, A 0.000, B 0.000, C 0.000 }
gfCNCPoint3[15979] = {X 256.0401, Y 47.4028, Z -4.6667, A 0.000, B 0.000, C 0.000 }
gfCNCPoint3[15980] = {X 255.6308, Y 46.4590, Z -4.6667, A 0.000, B 0.000, C 0.000 }
gfCNCPoint3[15981] = {X 255.4666, Y 45.7568, Z -4.6667, A 0.000, B 0.000, C 0.000 }
gfCNCPoint3[15982] = {X 255.4077, Y 45.0380, Z -4.6667, A 0.000, B 0.000, C 0.000 }
gfCNCPoint3[15983] = {X 255.4080, Y 44.1417, Z -4.6667, A 0.000, B 0.000, C 0.000 }
gfCNCPoint3[15984] = {X 255.5183, Y 43.1751, Z -4.6667, A 0.000, B 0.000, C 0.000 }
gfCNCPoint3[15985] = {X 255.8181, Y 42.2497, Z -4.6667, A 0.000, B 0.000, C 0.000 }
gfCNCPoint3[15986] = {X 256.2955, Y 41.4021, Z -4.6667, A 0.000, B 0.000, C 0.000 }
gfCNCPoint3[15987] = {X 256.9315, Y 40.6660, Z -4.6667, A 0.000, B 0.000, C 0.000 }
gfCNCPoint3[15988] = {X 256.9315, Y 35.0338, Z -4.6667, A 0.000, B 0.000, C 0.000 }
gfCNCPoint3[15989] = {X 255.1097, Y 35.0338, Z -4.6667, A 0.000, B 0.000, C 0.000 }
gfCNCPoint3[15990] = {X 251.0865, Y 42.8707, Z -4.6667, A 0.000, B 0.000, C 0.000 }
gfCNCPoint3[15991] = {X 251.2237, Y 43.5128, Z -4.6667, A 0.000, B 0.000, C 0.000 }
gfCNCPoint3[15992] = {X 251.2734, Y 44.1675, Z -4.6667, A 0.000, B 0.000, C 0.000 }
gfCNCPoint3[15993] = {X 251.2736, Y 45.0000, Z -4.6667, A 0.000, B 0.000, C 0.000 }
gfCNCPoint3[15994] = {X 251.2174, Y 45.7380, Z -4.6667, A 0.000, B 0.000, C 0.000 }
gfCNCPoint3[15995] = {X 251.0503, Y 46.4590, Z -4.6667, A 0.000, B 0.000, C 0.000 }
gfCNCPoint3[15996] = {X 250.6346, Y 47.4142, Z -4.6667, A 0.000, B 0.000, C 0.000 }
gfCNCPoint3[15997] = {X 250.0255, Y 48.2593, Z -4.6667, A 0.000, B 0.000, C 0.000 }
gfCNCPoint3[15998] = {X 249.2510, Y 48.9560, Z -4.6667, A 0.000, B 0.000, C 0.000 }
gfCNCPoint3[15999] = {X 248.3462, Y 49.4723, Z -4.6667, A 0.000, B 0.000, C 0.000 }
gfCNCPoint3[16000] = {X 247.3525, Y 49.7849, Z -4.6667, A 0.000, B 0.000, C 0.000 }
gfCNCPoint3[16001] = {X 246.8754, Y 49.8562, Z -4.6667, A 0.000, B 0.000, C 0.000 }
gfCNCPoint3[16002] = {X 246.3936, Y 49.8800, Z -4.6667, A 0.000, B 0.000, C 0.000 }
gfCNCPoint3[16003] = {X 242.5312, Y 49.8800, Z -4.6667, A 0.000, B 0.000, C 0.000 }
gfCNCPoint3[16004] = {X 242.5312, Y 49.4000, Z -4.6667, A 0.000, B 0.000, C 0.000 }
gfCNCPoint3[16005] = {X 239.8075, Y 49.4000, Z -4.6667, A 0.000, B 0.000, C 0.000 }
gfCNCPoint3[16006] = {X 238.8284, Y 49.2897, Z -4.6667, A 0.000, B 0.000, C 0.000 }
gfCNCPoint3[16007] = {X 237.8984, Y 48.9643, Z -4.6667, A 0.000, B 0.000, C 0.000 }
gfCNCPoint3[16008] = {X 237.0641, Y 48.4401, Z -4.6667, A 0.000, B 0.000, C 0.000 }
gfCNCPoint3[16009] = {X 236.3674, Y 47.7434, Z -4.6667, A 0.000, B 0.000, C 0.000 }
gfCNCPoint3[16010] = {X 235.8432, Y 46.9091, Z -4.6667, A 0.000, B 0.000, C 0.000 }
gfCNCPoint3[16011] = {X 235.5178, Y 45.9791, Z -4.6667, A 0.000, B 0.000, C 0.000 }
gfCNCPoint3[16012] = {X 235.4075, Y 45.0000, Z -4.6667, A 0.000, B 0.000, C 0.000 }
gfCNCPoint3[16013] = {X 235.4079, Y 44.1483, Z -4.6667, A 0.000, B 0.000, C 0.000 }
gfCNCPoint3[16014] = {X 235.5063, Y 43.2816, Z -4.6667, A 0.000, B 0.000, C 0.000 }
gfCNCPoint3[16015] = {X 235.7737, Y 42.4514, Z -4.6667, A 0.000, B 0.000, C 0.000 }
gfCNCPoint3[16016] = {X 236.1996, Y 41.6903, Z -4.6667, A 0.000, B 0.000, C 0.000 }
gfCNCPoint3[16017] = {X 236.7672, Y 41.0281, Z -4.6667, A 0.000, B 0.000, C 0.000 }
gfCNCPoint3[16018] = {X 237.4544, Y 40.4909, Z -4.6667, A 0.000, B 0.000, C 0.000 }
gfCNCPoint3[16019] = {X 238.2339, Y 40.0998, Z -4.6667, A 0.000, B 0.000, C 0.000 }
gfCNCPoint3[16020] = {X 242.1748, Y 32.3861, Z -4.6667, A 0.000, B 0.000, C 0.000 }
gfCNCPoint3[16021] = {X 241.0112, Y 31.5936, Z -4.6667, A 0.000, B 0.000, C 0.000 }
gfCNCPoint3[16022] = {X 239.9542, Y 30.6638, Z -4.6667, A 0.000, B 0.000, C 0.000 }
gfCNCPoint3[16023] = {X 239.0198, Y 29.6108, Z -4.6667, A 0.000, B 0.000, C 0.000 }
gfCNCPoint3[16024] = {X 238.2225, Y 28.4506, Z -4.6667, A 0.000, B 0.000, C 0.000 }
gfCNCPoint3[16025] = {X 237.5742, Y 27.2010, Z -4.6667, A 0.000, B 0.000, C 0.000 }
gfCNCPoint3[16026] = {X 237.0849, Y 25.8809, Z -4.6667, A 0.000, B 0.000, C 0.000 }
gfCNCPoint3[16027] = {X 236.6632, Y 24.0613, Z -4.6667, A 0.000, B 0.000, C 0.000 }
gfCNCPoint3[16028] = {X 236.4483, Y 22.2058, Z -4.6667, A 0.000, B 0.000, C 0.000 }
gfCNCPoint3[16029] = {X 236.4431, Y 20.3379, Z -4.6667, A 0.000, B 0.000, C 0.000 }
gfCNCPoint3[16030] = {X 236.6476, Y 18.4812, Z -4.6667, A 0.000, B 0.000, C 0.000 }
gfCNCPoint3[16031] = {X 237.0592, Y 16.6592, Z -4.6667, A 0.000, B 0.000, C 0.000 }
gfCNCPoint3[16032] = {X 237.6334, Y 15.0729, Z -4.6667, A 0.000, B 0.000, C 0.000 }
gfCNCPoint3[16033] = {X 238.4257, Y 13.5835, Z -4.6667, A 0.000, B 0.000, C 0.000 }
gfCNCPoint3[16034] = {X 239.4201, Y 12.2208, Z -4.6667, A 0.000, B 0.000, C 0.000 }
gfCNCPoint3[16035] = {X 240.5969, Y 11.0119, Z -4.6667, A 0.000, B 0.000, C 0.000 }
gfCNCPoint3[16036] = {X 241.9324, Y 9.9812, Z -4.6667, A 0.000, B 0.000, C 0.000 }
gfCNCPoint3[16037] = {X 243.4000, Y 9.1492, Z -4.6667, A 0.000, B 0.000, C 0.000 }
gfCNCPoint3[16038] = {X 244.9703, Y 8.5326, Z -4.6667, A 0.000, B 0.000, C 0.000 }
gfCNCPoint3[16039] = {X 246.6119, Y 8.1437, Z -4.6667, A 0.000, B 0.000, C 0.000 }
gfCNCPoint3[16040] = {X 248.7155, Y 7.8714, Z -4.6667, A 0.000, B 0.000, C 0.000 }
gfCNCPoint3[16041] = {X 250.8351, Y 7.7906, Z -4.6667, A 0.000, B 0.000, C 0.000 }
gfCNCPoint3[16042] = {X 266.7640, Y 7.7906, Z -4.6667, A 0.000, B 0.000, C 0.000 }
gfCNCPoint3[16043] = {X 267.7369, Y 7.9075, Z -4.6667, A 0.000, B 0.000, C 0.000 }
gfCNCPoint3[16044] = {X 268.6598, Y 8.2366, Z -4.6667, A 0.000, B 0.000, C 0.000 }
gfCNCPoint3[16045] = {X 269.4870, Y 8.7618, Z -4.6667, A 0.000, B 0.000, C 0.000 }
gfCNCPoint3[16046] = {X 270.1776, Y 9.4569, Z -4.6667, A 0.000, B 0.000, C 0.000 }
gfCNCPoint3[16047] = {X 270.6974, Y 10.2876, Z -4.6667, A 0.000, B 0.000, C 0.000 }
gfCNCPoint3[16048] = {X 271.0205, Y 11.2126, Z -4.6667, A 0.000, B 0.000, C 0.000 }
gfCNCPoint3[16049] = {X 271.1310, Y 12.1863, Z -4.6667, A 0.000, B 0.000, C 0.000 }
gfCNCPoint3[16050] = {X 271.1308, Y 13.0233, Z -4.6667, A 0.000, B 0.000, C 0.000 }
gfCNCPoint3[16051] = {X 271.0225, Y 13.9492, Z -4.6667, A 0.000, B 0.000, C 0.000 }
gfCNCPoint3[16052] = {X 270.7216, Y 14.8314, Z -4.6667, A 0.000, B 0.000, C 0.000 }
gfCNCPoint3[16053] = {X 270.2416, Y 15.6305, Z -4.6667, A 0.000, B 0.000, C 0.000 }
gfCNCPoint3[16054] = {X 269.6040, Y 16.3106, Z -4.6667, A 0.000, B 0.000, C 0.000 }
gfCNCPoint3[16055] = {X 269.6039, Y 40.8761, Z -4.6667, A 0.000, B 0.000, C 0.000 }
gfCNCPoint3[16056] = {X 270.2483, Y 41.5652, Z -4.6667, A 0.000, B 0.000, C 0.000 }
gfCNCPoint3[16057] = {X 270.7311, Y 42.3759, Z -4.6667, A 0.000, B 0.000, C 0.000 }
gfCNCPoint3[16058] = {X 271.0299, Y 43.2708, Z -4.6667, A 0.000, B 0.000, C 0.000 }
gfCNCPoint3[16059] = {X 271.1310, Y 44.2089, Z -4.6667, A 0.000, B 0.000, C 0.000 }
gfCNCPoint3[16060] = {X 271.1310, Y 45.0000, Z -4.6667, A 0.000, B 0.000, C 0.000 }
gfCNCPoint3[16061] = {X 271.0207, Y 45.9791, Z -4.6667, A 0.000, B 0.000, C 0.000 }
gfCNCPoint3[16062] = {X 270.6953, Y 46.9091, Z -4.6667, A 0.000, B 0.000, C 0.000 }
gfCNCPoint3[16063] = {X 270.1711, Y 47.7434, Z -4.6667, A 0.000, B 0.000, C 0.000 }
gfCNCPoint3[16064] = {X 269.4744, Y 48.4401, Z -4.6667, A 0.000, B 0.000, C 0.000 }
gfCNCPoint3[16065] = {X 268.6401, Y 48.9643, Z -4.6667, A 0.000, B 0.000, C 0.000 }
gfCNCPoint3[16066] = {X 267.7101, Y 49.2897, Z -4.6667, A 0.000, B 0.000, C 0.000 }
gfCNCPoint3[16067] = {X 266.7310, Y 49.4000, Z -4.6667, A 0.000, B 0.000, C 0.000 }
gfCNCPoint3[16068] = {X 260.2876, Y 49.4000, Z -4.6667, A 0.000, B 0.000, C 0.000 }
gfCNCPoint3[16069] = {X 259.3085, Y 49.2897, Z -4.6667, A 0.000, B 0.000, C 0.000 }
gfCNCPoint3[16070] = {X 258.3785, Y 48.9643, Z -4.6667, A 0.000, B 0.000, C 0.000 }
gfCNCPoint3[16071] = {X 257.5442, Y 48.4400, Z -4.6667, A 0.000, B 0.000, C 0.000 }
gfCNCPoint3[16072] = {X 256.8475, Y 47.7433, Z -4.6667, A 0.000, B 0.000, C 0.000 }
gfCNCPoint3[16073] = {X 256.3233, Y 46.9091, Z -4.6667, A 0.000, B 0.000, C 0.000 }
gfCNCPoint3[16074] = {X 255.9979, Y 45.9791, Z -4.6667, A 0.000, B 0.000, C 0.000 }
gfCNCPoint3[16075] = {X 255.8876, Y 45.0000, Z -4.6667, A 0.000, B 0.000, C 0.000 }
gfCNCPoint3[16076] = {X 255.8880, Y 44.1483, Z -4.6667, A 0.000, B 0.000, C 0.000 }
gfCNCPoint3[16077] = {X 255.9984, Y 43.2275, Z -4.6667, A 0.000, B 0.000, C 0.000 }
gfCNCPoint3[16078] = {X 256.2993, Y 42.3503, Z -4.6667, A 0.000, B 0.000, C 0.000 }
gfCNCPoint3[16079] = {X 256.7775, Y 41.5556, Z -4.6667, A 0.000, B 0.000, C 0.000 }
gfCNCPoint3[16080] = {X 257.4115, Y 40.8789, Z -4.6667, A 0.000, B 0.000, C 0.000 }
gfCNCPoint3[16081] = {X 257.4115, Y 34.5538, Z -4.6667, A 0.000, B 0.000, C 0.000 }
gfCNCPoint3[16082] = {X 254.8166, Y 34.5538, Z -4.6667, A 0.000, B 0.000, C 0.000 }
gfCNCPoint3[16083] = {X 250.5704, Y 42.8252, Z -4.6667, A 0.000, B 0.000, C 0.000 }
gfCNCPoint3[16084] = {X 250.7374, Y 43.5081, Z -4.6667, A 0.000, B 0.000, C 0.000 }
gfCNCPoint3[16085] = {X 250.7936, Y 44.2089, Z -4.6667, A 0.000, B 0.000, C 0.000 }
gfCNCPoint3[16086] = {X 250.7936, Y 45.0000, Z -4.6667, A 0.000, B 0.000, C 0.000 }
gfCNCPoint3[16087] = {X 250.6832, Y 45.9791, Z -4.6667, A 0.000, B 0.000, C 0.000 }
gfCNCPoint3[16088] = {X 250.3578, Y 46.9091, Z -4.6667, A 0.000, B 0.000, C 0.000 }
gfCNCPoint3[16089] = {X 249.8336, Y 47.7434, Z -4.6667, A 0.000, B 0.000, C 0.000 }
gfCNCPoint3[16090] = {X 249.1369, Y 48.4401, Z -4.6667, A 0.000, B 0.000, C 0.000 }
gfCNCPoint3[16091] = {X 248.3026, Y 48.9643, Z -4.6667, A 0.000, B 0.000, C 0.000 }
gfCNCPoint3[16092] = {X 247.3727, Y 49.2897, Z -4.6667, A 0.000, B 0.000, C 0.000 }
gfCNCPoint3[16093] = {X 246.3936, Y 49.4000, Z -4.6667, A 0.000, B 0.000, C 0.000 }
gfCNCPoint3[16094] = {X 242.5312, Y 49.4000, Z -4.6667, A 0.000, B 0.000, C 0.000 }
gfCNCPoint3[16095] = {X 242.5312, Y 49.8800, Z -4.6667, A 0.000, B 0.000, C 0.000 }
gfCNCPoint3[16096] = {X 243.4812, Y 50.5824, Z -4.6667, A 0.000, B 0.000, C 0.000 }
gfCNCPoint3[16097] = {X 244.3384, Y 51.3953, Z -4.6667, A 0.000, B 0.000, C 0.000 }
gfCNCPoint3[16098] = {X 245.0903, Y 52.3066, Z -4.6667, A 0.000, B 0.000, C 0.000 }
gfCNCPoint3[16099] = {X 245.7256, Y 53.3027, Z -4.6667, A 0.000, B 0.000, C 0.000 }
gfCNCPoint3[16100] = {X 245.9755, Y 53.7843, Z -4.6667, A 0.000, B 0.000, C 0.000 }
gfCNCPoint3[16101] = {X 246.1980, Y 54.2793, Z -4.6667, A 0.000, B 0.000, C 0.000 }
gfCNCPoint3[16102] = {X 250.0854, Y 55.7951, Z -4.6667, A 0.000, B 0.000, C 0.000 }
gfCNCPoint3[16103] = {X 267.2823, Y 62.6208, Z -4.6667, A 0.000, B 0.000, C 0.000 }
gfCNCPoint3[16104] = {X 266.8843, Y 61.4461, Z -4.6667, A 0.000, B 0.000, C 0.000 }
gfCNCPoint3[16105] = {X 266.6399, Y 60.2302, Z -4.6667, A 0.000, B 0.000, C 0.000 }
gfCNCPoint3[16106] = {X 266.5529, Y 58.9930, Z -4.6667, A 0.000, B 0.000, C 0.000 }
gfCNCPoint3[16107] = {X 266.5527, Y 58.0000, Z -4.6667, A 0.000, B 0.000, C 0.000 }
gfCNCPoint3[16108] = {X 266.6262, Y 56.8093, Z -4.6667, A 0.000, B 0.000, C 0.000 }
gfCNCPoint3[16109] = {X 266.8456, Y 55.6367, Z -4.6667, A 0.000, B 0.000, C 0.000 }
gfCNCPoint3[16110] = {X 267.2076, Y 54.5000, Z -4.6667, A 0.000, B 0.000, C 0.000 }
gfCNCPoint3[16111] = {X 267.7067, Y 53.4164, Z -4.6667, A 0.000, B 0.000, C 0.000 }
gfCNCPoint3[16112] = {X 268.4728, Y 52.2132, Z -4.6667, A 0.000, B 0.000, C 0.000 }
gfCNCPoint3[16113] = {X 269.4075, Y 51.1357, Z -4.6667, A 0.000, B 0.000, C 0.000 }
gfCNCPoint3[16114] = {X 270.4903, Y 50.2072, Z -4.6667, A 0.000, B 0.000, C 0.000 }
gfCNCPoint3[16115] = {X 271.6979, Y 49.4479, Z -4.6667, A 0.000, B 0.000, C 0.000 }
gfCNCPoint3[16116] = {X 273.0039, Y 48.8744, Z -4.6667, A 0.000, B 0.000, C 0.000 }
gfCNCPoint3[16117] = {X 274.3800, Y 48.4989, Z -4.6667, A 0.000, B 0.000, C 0.000 }
gfCNCPoint3[16118] = {X 275.3020, Y 48.3648, Z -4.6667, A 0.000, B 0.000, C 0.000 }
gfCNCPoint3[16119] = {X 276.2327, Y 48.3200, Z -4.6667, A 0.000, B 0.000, C 0.000 }
gfCNCPoint3[16120] = {X 281.0411, Y 48.3200, Z -4.6667, A 0.000, B 0.000, C 0.000 }
gfCNCPoint3[16121] = {X 280.4347, Y 47.5134, Z -4.6667, A 0.000, B 0.000, C 0.000 }
gfCNCPoint3[16122] = {X 280.0072, Y 46.5992, Z -4.6667, A 0.000, B 0.000, C 0.000 }
gfCNCPoint3[16123] = {X 279.7768, Y 45.6167, Z -4.6667, A 0.000, B 0.000, C 0.000 }
gfCNCPoint3[16124] = {X 279.7488, Y 45.3288, Z -4.6667, A 0.000, B 0.000, C 0.000 }
gfCNCPoint3[16125] = {X 279.7378, Y 45.0398, Z -4.6667, A 0.000, B 0.000, C 0.000 }
gfCNCPoint3[16126] = {X 279.7377, Y 44.2043, Z -4.6667, A 0.000, B 0.000, C 0.000 }
gfCNCPoint3[16127] = {X 279.8420, Y 43.2207, Z -4.6667, A 0.000, B 0.000, C 0.000 }
gfCNCPoint3[16128] = {X 280.1406, Y 42.2777, Z -4.6667, A 0.000, B 0.000, C 0.000 }
gfCNCPoint3[16129] = {X 280.6215, Y 41.4134, Z -4.6667, A 0.000, B 0.000, C 0.000 }
gfCNCPoint3[16130] = {X 281.2653, Y 40.6624, Z -4.6667, A 0.000, B 0.000, C 0.000 }
gfCNCPoint3[16131] = {X 281.2649, Y 16.5239, Z -4.6667, A 0.000, B 0.000, C 0.000 }
gfCNCPoint3[16132] = {X 280.6239, Y 15.7823, Z -4.6667, A 0.000, B 0.000, C 0.000 }
gfCNCPoint3[16133] = {X 280.1440, Y 14.9276, Z -4.6667, A 0.000, B 0.000, C 0.000 }
gfCNCPoint3[16134] = {X 279.8446, Y 13.9942, Z -4.6667, A 0.000, B 0.000, C 0.000 }
gfCNCPoint3[16135] = {X 279.7378, Y 13.0198, Z -4.6667, A 0.000, B 0.000, C 0.000 }
gfCNCPoint3[16136] = {X 279.7377, Y 12.1868, Z -4.6667, A 0.000, B 0.000, C 0.000 }
gfCNCPoint3[16137] = {X 279.8242, Y 11.2717, Z -4.6667, A 0.000, B 0.000, C 0.000 }
gfCNCPoint3[16138] = {X 280.0809, Y 10.3891, Z -4.6667, A 0.000, B 0.000, C 0.000 }
gfCNCPoint3[16139] = {X 280.5256, Y 9.5280, Z -4.6667, A 0.000, B 0.000, C 0.000 }
gfCNCPoint3[16140] = {X 281.1317, Y 8.7718, Z -4.6667, A 0.000, B 0.000, C 0.000 }
gfCNCPoint3[16141] = {X 281.8753, Y 8.1503, Z -4.6667, A 0.000, B 0.000, C 0.000 }
gfCNCPoint3[16142] = {X 282.7270, Y 7.6879, Z -4.6667, A 0.000, B 0.000, C 0.000 }
gfCNCPoint3[16143] = {X 283.6533, Y 7.4030, Z -4.6667, A 0.000, B 0.000, C 0.000 }
gfCNCPoint3[16144] = {X 284.6177, Y 7.3068, Z -4.6667, A 0.000, B 0.000, C 0.000 }
gfCNCPoint3[16145] = {X 291.0611, Y 7.3068, Z -4.6667, A 0.000, B 0.000, C 0.000 }
gfCNCPoint3[16146] = {X 292.0255, Y 7.4030, Z -4.6667, A 0.000, B 0.000, C 0.000 }
gfCNCPoint3[16147] = {X 292.9518, Y 7.6879, Z -4.6667, A 0.000, B 0.000, C 0.000 }
gfCNCPoint3[16148] = {X 293.8035, Y 8.1503, Z -4.6667, A 0.000, B 0.000, C 0.000 }
gfCNCPoint3[16149] = {X 294.5471, Y 8.7718, Z -4.6667, A 0.000, B 0.000, C 0.000 }
gfCNCPoint3[16150] = {X 295.1532, Y 9.5280, Z -4.6667, A 0.000, B 0.000, C 0.000 }
gfCNCPoint3[16151] = {X 295.5979, Y 10.3891, Z -4.6667, A 0.000, B 0.000, C 0.000 }
gfCNCPoint3[16152] = {X 295.8044, Y 11.0397, Z -4.6667, A 0.000, B 0.000, C 0.000 }
gfCNCPoint3[16153] = {X 295.9181, Y 11.7127, Z -4.6667, A 0.000, B 0.000, C 0.000 }
gfCNCPoint3[16154] = {X 295.9354, Y 11.9495, Z -4.6667, A 0.000, B 0.000, C 0.000 }
gfCNCPoint3[16155] = {X 295.9411, Y 12.1868, Z -4.6667, A 0.000, B 0.000, C 0.000 }
gfCNCPoint3[16156] = {X 295.9409, Y 13.0237, Z -4.6667, A 0.000, B 0.000, C 0.000 }
gfCNCPoint3[16157] = {X 295.9342, Y 13.2382, Z -4.6667, A 0.000, B 0.000, C 0.000 }
gfCNCPoint3[16158] = {X 295.9180, Y 13.4521, Z -4.6667, A 0.000, B 0.000, C 0.000 }
gfCNCPoint3[16159] = {X 298.3067, Y 13.6853, Z -4.6667, A 0.000, B 0.000, C 0.000 }
gfCNCPoint3[16160] = {X 298.1361, Y 14.6936, Z -4.6667, A 0.000, B 0.000, C 0.000 }
gfCNCPoint3[16161] = {X 297.8259, Y 15.6681, Z -4.6667, A 0.000, B 0.000, C 0.000 }
gfCNCPoint3[16162] = {X 297.3822, Y 16.5894, Z -4.6667, A 0.000, B 0.000, C 0.000 }
gfCNCPoint3[16163] = {X 296.8138, Y 17.4396, Z -4.6667, A 0.000, B 0.000, C 0.000 }
gfCNCPoint3[16164] = {X 296.8141, Y 19.2365, Z -4.6667, A 0.000, B 0.000, C 0.000 }
gfCNCPoint3[16165] = {X 299.7992, Y 19.2365, Z -4.6667, A 0.000, B 0.000, C 0.000 }
gfCNCPoint3[16166] = {X 299.7993, Y 17.4392, Z -4.6667, A 0.000, B 0.000, C 0.000 }
gfCNCPoint3[16167] = {X 299.2310, Y 16.5891, Z -4.6667, A 0.000, B 0.000, C 0.000 }
gfCNCPoint3[16168] = {X 298.7874, Y 15.6678, Z -4.6667, A 0.000, B 0.000, C 0.000 }
gfCNCPoint3[16169] = {X 298.4773, Y 14.6935, Z -4.6667, A 0.000, B 0.000, C 0.000 }
gfCNCPoint3[16170] = {X 298.3067, Y 13.6853, Z -4.6667, A 0.000, B 0.000, C 0.000 }
gfCNCPoint3[16171] = {X 295.9180, Y 13.4521, Z -4.6667, A 0.000, B 0.000, C 0.000 }
gfCNCPoint3[16172] = {X 295.7560, Y 14.3095, Z -4.6667, A 0.000, B 0.000, C 0.000 }
gfCNCPoint3[16173] = {X 295.4438, Y 15.1243, Z -4.6667, A 0.000, B 0.000, C 0.000 }
gfCNCPoint3[16174] = {X 294.9915, Y 15.8705, Z -4.6667, A 0.000, B 0.000, C 0.000 }
gfCNCPoint3[16175] = {X 294.4136, Y 16.5242, Z -4.6667, A 0.000, B 0.000, C 0.000 }
gfCNCPoint3[16176] = {X 294.4146, Y 21.6365, Z -4.6667, A 0.000, B 0.000, C 0.000 }
gfCNCPoint3[16177] = {X 302.1990, Y 21.6365, Z -4.6667, A 0.000, B 0.000, C 0.000 }
gfCNCPoint3[16178] = {X 302.1994, Y 16.5238, Z -4.6667, A 0.000, B 0.000, C 0.000 }
gfCNCPoint3[16179] = {X 301.6216, Y 15.8701, Z -4.6667, A 0.000, B 0.000, C 0.000 }
gfCNCPoint3[16180] = {X 301.1694, Y 15.1240, Z -4.6667, A 0.000, B 0.000, C 0.000 }
gfCNCPoint3[16181] = {X 300.8574, Y 14.3094, Z -4.6667, A 0.000, B 0.000, C 0.000 }
gfCNCPoint3[16182] = {X 300.6953, Y 13.4521, Z -4.6667, A 0.000, B 0.000, C 0.000 }
gfCNCPoint3[16183] = {X 300.6791, Y 13.2371, Z -4.6667, A 0.000, B 0.000, C 0.000 }
gfCNCPoint3[16184] = {X 300.6724, Y 13.0215, Z -4.6667, A 0.000, B 0.000, C 0.000 }
gfCNCPoint3[16185] = {X 300.6723, Y 12.1868, Z -4.6667, A 0.000, B 0.000, C 0.000 }
gfCNCPoint3[16186] = {X 300.6780, Y 11.9495, Z -4.6667, A 0.000, B 0.000, C 0.000 }
gfCNCPoint3[16187] = {X 300.6953, Y 11.7127, Z -4.6667, A 0.000, B 0.000, C 0.000 }
gfCNCPoint3[16188] = {X 300.8090, Y 11.0397, Z -4.6667, A 0.000, B 0.000, C 0.000 }
gfCNCPoint3[16189] = {X 301.0154, Y 10.3891, Z -4.6667, A 0.000, B 0.000, C 0.000 }
gfCNCPoint3[16190] = {X 301.4602, Y 9.5280, Z -4.6667, A 0.000, B 0.000, C 0.000 }
gfCNCPoint3[16191] = {X 302.0663, Y 8.7718, Z -4.6667, A 0.000, B 0.000, C 0.000 }
gfCNCPoint3[16192] = {X 302.8099, Y 8.1503, Z -4.6667, A 0.000, B 0.000, C 0.000 }
gfCNCPoint3[16193] = {X 303.6616, Y 7.6879, Z -4.6667, A 0.000, B 0.000, C 0.000 }
gfCNCPoint3[16194] = {X 304.5879, Y 7.4030, Z -4.6667, A 0.000, B 0.000, C 0.000 }
gfCNCPoint3[16195] = {X 305.5523, Y 7.3068, Z -4.6667, A 0.000, B 0.000, C 0.000 }
gfCNCPoint3[16196] = {X 311.9957, Y 7.3068, Z -4.6667, A 0.000, B 0.000, C 0.000 }
gfCNCPoint3[16197] = {X 312.9478, Y 7.4006, Z -4.6667, A 0.000, B 0.000, C 0.000 }
gfCNCPoint3[16198] = {X 313.8632, Y 7.6783, Z -4.6667, A 0.000, B 0.000, C 0.000 }
gfCNCPoint3[16199] = {X 314.7069, Y 8.1292, Z -4.6667, A 0.000, B 0.000, C 0.000 }
gfCNCPoint3[16200] = {X 315.4464, Y 8.7361, Z -4.6667, A 0.000, B 0.000, C 0.000 }
gfCNCPoint3[16201] = {X 316.0533, Y 9.4756, Z -4.6667, A 0.000, B 0.000, C 0.000 }
gfCNCPoint3[16202] = {X 316.5043, Y 10.3193, Z -4.6667, A 0.000, B 0.000, C 0.000 }
gfCNCPoint3[16203] = {X 316.7820, Y 11.2348, Z -4.6667, A 0.000, B 0.000, C 0.000 }
gfCNCPoint3[16204] = {X 316.8757, Y 12.1868, Z -4.6667, A 0.000, B 0.000, C 0.000 }
gfCNCPoint3[16205] = {X 316.8755, Y 13.0237, Z -4.6667, A 0.000, B 0.000, C 0.000 }
gfCNCPoint3[16206] = {X 316.7682, Y 13.9967, Z -4.6667, A 0.000, B 0.000, C 0.000 }
gfCNCPoint3[16207] = {X 316.4689, Y 14.9287, Z -4.6667, A 0.000, B 0.000, C 0.000 }
gfCNCPoint3[16208] = {X 315.9895, Y 15.7823, Z -4.6667, A 0.000, B 0.000, C 0.000 }
gfCNCPoint3[16209] = {X 315.3495, Y 16.5230, Z -4.6667, A 0.000, B 0.000, C 0.000 }
gfCNCPoint3[16210] = {X 315.3481, Y 40.6625, Z -4.6667, A 0.000, B 0.000, C 0.000 }
gfCNCPoint3[16211] = {X 315.9892, Y 41.4041, Z -4.6667, A 0.000, B 0.000, C 0.000 }
gfCNCPoint3[16212] = {X 316.4692, Y 42.2587, Z -4.6667, A 0.000, B 0.000, C 0.000 }
gfCNCPoint3[16213] = {X 316.7686, Y 43.1921, Z -4.6667, A 0.000, B 0.000, C 0.000 }
gfCNCPoint3[16214] = {X 316.8755, Y 44.1664, Z -4.6667, A 0.000, B 0.000, C 0.000 }
gfCNCPoint3[16215] = {X 316.8757, Y 45.0000, Z -4.6667, A 0.000, B 0.000, C 0.000 }
gfCNCPoint3[16216] = {X 316.8749, Y 45.0899, Z -4.6667, A 0.000, B 0.000, C 0.000 }
gfCNCPoint3[16217] = {X 316.8724, Y 45.1799, Z -4.6667, A 0.000, B 0.000, C 0.000 }
gfCNCPoint3[16218] = {X 316.8594, Y 45.3987, Z -4.6667, A 0.000, B 0.000, C 0.000 }
gfCNCPoint3[16219] = {X 316.8366, Y 45.6167, Z -4.6667, A 0.000, B 0.000, C 0.000 }
gfCNCPoint3[16220] = {X 316.6062, Y 46.5992, Z -4.6667, A 0.000, B 0.000, C 0.000 }
gfCNCPoint3[16221] = {X 316.1787, Y 47.5134, Z -4.6667, A 0.000, B 0.000, C 0.000 }
gfCNCPoint3[16222] = {X 315.5723, Y 48.3200, Z -4.6667, A 0.000, B 0.000, C 0.000 }
gfCNCPoint3[16223] = {X 315.2205, Y 47.9934, Z -4.6667, A 0.000, B 0.000, C 0.000 }
gfCNCPoint3[16224] = {X 314.5413, Y 48.5889, Z -4.6667, A 0.000, B 0.000, C 0.000 }
gfCNCPoint3[16225] = {X 313.7548, Y 49.0331, Z -4.6667, A 0.000, B 0.000, C 0.000 }
gfCNCPoint3[16226] = {X 312.8942, Y 49.3073, Z -4.6667, A 0.000, B 0.000, C 0.000 }
gfCNCPoint3[16227] = {X 311.9957, Y 49.4000, Z -4.6667, A 0.000, B 0.000, C 0.000 }
gfCNCPoint3[16228] = {X 305.5523, Y 49.4000, Z -4.6667, A 0.000, B 0.000, C 0.000 }
gfCNCPoint3[16229] = {X 304.5732, Y 49.2897, Z -4.6667, A 0.000, B 0.000, C 0.000 }
gfCNCPoint3[16230] = {X 303.6432, Y 48.9643, Z -4.6667, A 0.000, B 0.000, C 0.000 }
gfCNCPoint3[16231] = {X 302.8089, Y 48.4400, Z -4.6667, A 0.000, B 0.000, C 0.000 }
gfCNCPoint3[16232] = {X 302.1122, Y 47.7433, Z -4.6667, A 0.000, B 0.000, C 0.000 }
gfCNCPoint3[16233] = {X 301.5880, Y 46.9091, Z -4.6667, A 0.000, B 0.000, C 0.000 }
gfCNCPoint3[16234] = {X 301.2626, Y 45.9791, Z -4.6667, A 0.000, B 0.000, C 0.000 }
gfCNCPoint3[16235] = {X 301.1523, Y 45.0000, Z -4.6667, A 0.000, B 0.000, C 0.000 }
gfCNCPoint3[16236] = {X 301.1524, Y 44.1993, Z -4.6667, A 0.000, B 0.000, C 0.000 }
gfCNCPoint3[16237] = {X 301.2700, Y 43.2559, Z -4.6667, A 0.000, B 0.000, C 0.000 }
gfCNCPoint3[16238] = {X 301.5730, Y 42.3547, Z -4.6667, A 0.000, B 0.000, C 0.000 }
gfCNCPoint3[16239] = {X 302.0493, Y 41.5318, Z -4.6667, A 0.000, B 0.000, C 0.000 }
gfCNCPoint3[16240] = {X 302.6797, Y 40.8202, Z -4.6667, A 0.000, B 0.000, C 0.000 }
gfCNCPoint3[16241] = {X 302.6797, Y 34.1143, Z -4.6667, A 0.000, B 0.000, C 0.000 }
gfCNCPoint3[16242] = {X 293.9345, Y 34.1143, Z -4.6667, A 0.000, B 0.000, C 0.000 }
gfCNCPoint3[16243] = {X 293.9337, Y 40.8660, Z -4.6667, A 0.000, B 0.000, C 0.000 }
gfCNCPoint3[16244] = {X 294.5737, Y 41.5610, Z -4.6667, A 0.000, B 0.000, C 0.000 }
gfCNCPoint3[16245] = {X 295.0544, Y 42.3743, Z -4.6667, A 0.000, B 0.000, C 0.000 }
gfCNCPoint3[16246] = {X 295.3546, Y 43.2701, Z -4.6667, A 0.000, B 0.000, C 0.000 }
gfCNCPoint3[16247] = {X 295.4611, Y 44.2089, Z -4.6667, A 0.000, B 0.000, C 0.000 }
gfCNCPoint3[16248] = {X 295.4611, Y 45.0000, Z -4.6667, A 0.000, B 0.000, C 0.000 }
gfCNCPoint3[16249] = {X 295.3508, Y 45.9791, Z -4.6667, A 0.000, B 0.000, C 0.000 }
gfCNCPoint3[16250] = {X 295.0254, Y 46.9091, Z -4.6667, A 0.000, B 0.000, C 0.000 }
gfCNCPoint3[16251] = {X 294.5012, Y 47.7434, Z -4.6667, A 0.000, B 0.000, C 0.000 }
gfCNCPoint3[16252] = {X 293.8045, Y 48.4401, Z -4.6667, A 0.000, B 0.000, C 0.000 }
gfCNCPoint3[16253] = {X 292.9702, Y 48.9643, Z -4.6667, A 0.000, B 0.000, C 0.000 }
gfCNCPoint3[16254] = {X 292.0402, Y 49.2897, Z -4.6667, A 0.000, B 0.000, C 0.000 }
gfCNCPoint3[16255] = {X 291.0611, Y 49.4000, Z -4.6667, A 0.000, B 0.000, C 0.000 }
gfCNCPoint3[16256] = {X 284.6177, Y 49.4000, Z -4.6667, A 0.000, B 0.000, C 0.000 }
gfCNCPoint3[16257] = {X 283.6386, Y 49.2897, Z -4.6667, A 0.000, B 0.000, C 0.000 }
gfCNCPoint3[16258] = {X 282.7086, Y 48.9643, Z -4.6667, A 0.000, B 0.000, C 0.000 }
gfCNCPoint3[16259] = {X 281.8743, Y 48.4400, Z -4.6667, A 0.000, B 0.000, C 0.000 }
gfCNCPoint3[16260] = {X 281.1776, Y 47.7433, Z -4.6667, A 0.000, B 0.000, C 0.000 }
gfCNCPoint3[16261] = {X 280.6534, Y 46.9091, Z -4.6667, A 0.000, B 0.000, C 0.000 }
gfCNCPoint3[16262] = {X 280.3280, Y 45.9791, Z -4.6667, A 0.000, B 0.000, C 0.000 }
gfCNCPoint3[16263] = {X 280.2177, Y 45.0000, Z -4.6667, A 0.000, B 0.000, C 0.000 }
gfCNCPoint3[16264] = {X 280.2177, Y 44.2068, Z -4.6667, A 0.000, B 0.000, C 0.000 }
gfCNCPoint3[16265] = {X 280.3224, Y 43.2698, Z -4.6667, A 0.000, B 0.000, C 0.000 }
gfCNCPoint3[16266] = {X 280.6223, Y 42.3759, Z -4.6667, A 0.000, B 0.000, C 0.000 }
gfCNCPoint3[16267] = {X 281.1038, Y 41.5652, Z -4.6667, A 0.000, B 0.000, C 0.000 }
gfCNCPoint3[16268] = {X 281.7453, Y 40.8743, Z -4.6667, A 0.000, B 0.000, C 0.000 }
gfCNCPoint3[16269] = {X 281.7449, Y 16.3108, Z -4.6667, A 0.000, B 0.000, C 0.000 }
gfCNCPoint3[16270] = {X 281.1004, Y 15.6217, Z -4.6667, A 0.000, B 0.000, C 0.000 }
gfCNCPoint3[16271] = {X 280.6176, Y 14.8110, Z -4.6667, A 0.000, B 0.000, C 0.000 }
gfCNCPoint3[16272] = {X 280.3188, Y 13.9160, Z -4.6667, A 0.000, B 0.000, C 0.000 }
gfCNCPoint3[16273] = {X 280.2177, Y 12.9779, Z -4.6667, A 0.000, B 0.000, C 0.000 }
gfCNCPoint3[16274] = {X 280.2177, Y 12.1868, Z -4.6667, A 0.000, B 0.000, C 0.000 }
gfCNCPoint3[16275] = {X 280.3280, Y 11.2077, Z -4.6667, A 0.000, B 0.000, C 0.000 }
gfCNCPoint3[16276] = {X 280.6534, Y 10.2777, Z -4.6667, A 0.000, B 0.000, C 0.000 }
gfCNCPoint3[16277] = {X 281.1776, Y 9.4435, Z -4.6667, A 0.000, B 0.000, C 0.000 }
gfCNCPoint3[16278] = {X 281.8743, Y 8.7468, Z -4.6667, A 0.000, B 0.000, C 0.000 }
gfCNCPoint3[16279] = {X 282.7086, Y 8.2226, Z -4.6667, A 0.000, B 0.000, C 0.000 }
gfCNCPoint3[16280] = {X 283.6386, Y 7.8971, Z -4.6667, A 0.000, B 0.000, C 0.000 }
gfCNCPoint3[16281] = {X 284.6177, Y 7.7868, Z -4.6667, A 0.000, B 0.000, C 0.000 }
gfCNCPoint3[16282] = {X 291.0611, Y 7.7868, Z -4.6667, A 0.000, B 0.000, C 0.000 }
gfCNCPoint3[16283] = {X 292.0402, Y 7.8971, Z -4.6667, A 0.000, B 0.000, C 0.000 }
gfCNCPoint3[16284] = {X 292.9702, Y 8.2226, Z -4.6667, A 0.000, B 0.000, C 0.000 }
gfCNCPoint3[16285] = {X 293.8045, Y 8.7468, Z -4.6667, A 0.000, B 0.000, C 0.000 }
gfCNCPoint3[16286] = {X 294.5012, Y 9.4435, Z -4.6667, A 0.000, B 0.000, C 0.000 }
gfCNCPoint3[16287] = {X 295.0254, Y 10.2777, Z -4.6667, A 0.000, B 0.000, C 0.000 }
gfCNCPoint3[16288] = {X 295.3508, Y 11.2077, Z -4.6667, A 0.000, B 0.000, C 0.000 }
gfCNCPoint3[16289] = {X 295.4611, Y 12.1868, Z -4.6667, A 0.000, B 0.000, C 0.000 }
gfCNCPoint3[16290] = {X 295.4609, Y 13.0233, Z -4.6667, A 0.000, B 0.000, C 0.000 }
gfCNCPoint3[16291] = {X 295.3526, Y 13.9494, Z -4.6667, A 0.000, B 0.000, C 0.000 }
gfCNCPoint3[16292] = {X 295.0516, Y 14.8318, Z -4.6667, A 0.000, B 0.000, C 0.000 }
gfCNCPoint3[16293] = {X 294.5714, Y 15.6310, Z -4.6667, A 0.000, B 0.000, C 0.000 }
gfCNCPoint3[16294] = {X 293.9336, Y 16.3110, Z -4.6667, A 0.000, B 0.000, C 0.000 }
gfCNCPoint3[16295] = {X 293.9347, Y 22.1165, Z -4.6667, A 0.000, B 0.000, C 0.000 }
gfCNCPoint3[16296] = {X 302.6790, Y 22.1165, Z -4.6667, A 0.000, B 0.000, C 0.000 }
gfCNCPoint3[16297] = {X 302.6794, Y 16.3107, Z -4.6667, A 0.000, B 0.000, C 0.000 }
gfCNCPoint3[16298] = {X 302.0349, Y 15.6216, Z -4.6667, A 0.000, B 0.000, C 0.000 }
gfCNCPoint3[16299] = {X 301.5522, Y 14.8109, Z -4.6667, A 0.000, B 0.000, C 0.000 }
gfCNCPoint3[16300] = {X 301.2534, Y 13.9160, Z -4.6667, A 0.000, B 0.000, C 0.000 }
gfCNCPoint3[16301] = {X 301.1523, Y 12.9779, Z -4.6667, A 0.000, B 0.000, C 0.000 }
gfCNCPoint3[16302] = {X 301.1523, Y 12.1868, Z -4.6667, A 0.000, B 0.000, C 0.000 }
gfCNCPoint3[16303] = {X 301.2626, Y 11.2077, Z -4.6667, A 0.000, B 0.000, C 0.000 }
gfCNCPoint3[16304] = {X 301.5880, Y 10.2777, Z -4.6667, A 0.000, B 0.000, C 0.000 }
gfCNCPoint3[16305] = {X 302.1122, Y 9.4435, Z -4.6667, A 0.000, B 0.000, C 0.000 }
gfCNCPoint3[16306] = {X 302.8089, Y 8.7468, Z -4.6667, A 0.000, B 0.000, C 0.000 }
gfCNCPoint3[16307] = {X 303.6432, Y 8.2226, Z -4.6667, A 0.000, B 0.000, C 0.000 }
gfCNCPoint3[16308] = {X 304.5732, Y 7.8971, Z -4.6667, A 0.000, B 0.000, C 0.000 }
gfCNCPoint3[16309] = {X 305.5523, Y 7.7868, Z -4.6667, A 0.000, B 0.000, C 0.000 }
gfCNCPoint3[16310] = {X 311.9957, Y 7.7868, Z -4.6667, A 0.000, B 0.000, C 0.000 }
gfCNCPoint3[16311] = {X 312.9748, Y 7.8971, Z -4.6667, A 0.000, B 0.000, C 0.000 }
gfCNCPoint3[16312] = {X 313.9048, Y 8.2226, Z -4.6667, A 0.000, B 0.000, C 0.000 }
gfCNCPoint3[16313] = {X 314.7391, Y 8.7468, Z -4.6667, A 0.000, B 0.000, C 0.000 }
gfCNCPoint3[16314] = {X 315.4358, Y 9.4435, Z -4.6667, A 0.000, B 0.000, C 0.000 }
gfCNCPoint3[16315] = {X 315.9600, Y 10.2777, Z -4.6667, A 0.000, B 0.000, C 0.000 }
gfCNCPoint3[16316] = {X 316.2854, Y 11.2077, Z -4.6667, A 0.000, B 0.000, C 0.000 }
gfCNCPoint3[16317] = {X 316.3957, Y 12.1868, Z -4.6667, A 0.000, B 0.000, C 0.000 }
gfCNCPoint3[16318] = {X 316.3955, Y 13.0233, Z -4.6667, A 0.000, B 0.000, C 0.000 }
gfCNCPoint3[16319] = {X 316.2873, Y 13.9489, Z -4.6667, A 0.000, B 0.000, C 0.000 }
gfCNCPoint3[16320] = {X 315.9865, Y 14.8310, Z -4.6667, A 0.000, B 0.000, C 0.000 }
gfCNCPoint3[16321] = {X 315.5068, Y 15.6299, Z -4.6667, A 0.000, B 0.000, C 0.000 }
gfCNCPoint3[16322] = {X 314.8695, Y 16.3099, Z -4.6667, A 0.000, B 0.000, C 0.000 }
gfCNCPoint3[16323] = {X 314.8681, Y 40.8757, Z -4.6667, A 0.000, B 0.000, C 0.000 }
gfCNCPoint3[16324] = {X 315.5128, Y 41.5649, Z -4.6667, A 0.000, B 0.000, C 0.000 }
gfCNCPoint3[16325] = {X 315.9956, Y 42.3756, Z -4.6667, A 0.000, B 0.000, C 0.000 }
gfCNCPoint3[16326] = {X 316.2946, Y 43.2707, Z -4.6667, A 0.000, B 0.000, C 0.000 }
gfCNCPoint3[16327] = {X 316.3957, Y 44.2089, Z -4.6667, A 0.000, B 0.000, C 0.000 }
gfCNCPoint3[16328] = {X 316.3957, Y 45.0000, Z -4.6667, A 0.000, B 0.000, C 0.000 }
gfCNCPoint3[16329] = {X 316.3190, Y 45.8182, Z -4.6667, A 0.000, B 0.000, C 0.000 }
gfCNCPoint3[16330] = {X 316.0914, Y 46.6079, Z -4.6667, A 0.000, B 0.000, C 0.000 }
gfCNCPoint3[16331] = {X 315.7209, Y 47.3415, Z -4.6667, A 0.000, B 0.000, C 0.000 }
gfCNCPoint3[16332] = {X 315.2205, Y 47.9934, Z -4.6667, A 0.000, B 0.000, C 0.000 }
gfCNCPoint3[16333] = {X 315.5723, Y 48.3200, Z -4.6667, A 0.000, B 0.000, C 0.000 }
gfCNCPoint3[16334] = {X 324.3107, Y 48.3200, Z -4.6667, A 0.000, B 0.000, C 0.000 }
gfCNCPoint3[16335] = {X 325.5555, Y 48.4004, Z -4.6667, A 0.000, B 0.000, C 0.000 }
gfCNCPoint3[16336] = {X 326.7797, Y 48.6402, Z -4.6667, A 0.000, B 0.000, C 0.000 }
gfCNCPoint3[16337] = {X 325.5882, Y 48.0963, Z -4.6667, A 0.000, B 0.000, C 0.000 }
gfCNCPoint3[16338] = {X 324.4810, Y 47.3966, Z -4.6667, A 0.000, B 0.000, C 0.000 }
gfCNCPoint3[16339] = {X 323.4784, Y 46.5538, Z -4.6667, A 0.000, B 0.000, C 0.000 }
gfCNCPoint3[16340] = {X 322.8382, Y 45.9295, Z -4.6667, A 0.000, B 0.000, C 0.000 }
gfCNCPoint3[16341] = {X 322.2180, Y 45.2650, Z -4.6667, A 0.000, B 0.000, C 0.000 }
gfCNCPoint3[16342] = {X 321.6628, Y 44.5452, Z -4.6667, A 0.000, B 0.000, C 0.000 }
gfCNCPoint3[16343] = {X 323.6300, Y 43.1703, Z -4.6667, A 0.000, B 0.000, C 0.000 }
gfCNCPoint3[16344] = {X 323.0063, Y 42.0918, Z -4.6667, A 0.000, B 0.000, C 0.000 }
gfCNCPoint3[16345] = {X 322.5757, Y 40.9227, Z -4.6667, A 0.000, B 0.000, C 0.000 }
gfCNCPoint3[16346] = {X 322.3506, Y 39.6973, Z -4.6667, A 0.000, B 0.000, C 0.000 }
gfCNCPoint3[16347] = {X 322.3379, Y 38.4514, Z -4.6667, A 0.000, B 0.000, C 0.000 }
gfCNCPoint3[16348] = {X 322.5377, Y 37.2217, Z -4.6667, A 0.000, B 0.000, C 0.000 }
gfCNCPoint3[16349] = {X 322.9443, Y 36.0440, Z -4.6667, A 0.000, B 0.000, C 0.000 }
gfCNCPoint3[16350] = {X 323.5458, Y 34.9529, Z -4.6667, A 0.000, B 0.000, C 0.000 }
gfCNCPoint3[16351] = {X 327.7841, Y 28.6156, Z -4.6667, A 0.000, B 0.000, C 0.000 }
gfCNCPoint3[16352] = {X 328.5201, Y 27.6905, Z -4.6667, A 0.000, B 0.000, C 0.000 }
gfCNCPoint3[16353] = {X 329.3960, Y 26.8967, Z -4.6667, A 0.000, B 0.000, C 0.000 }
gfCNCPoint3[16354] = {X 330.3889, Y 26.2552, Z -4.6667, A 0.000, B 0.000, C 0.000 }
gfCNCPoint3[16355] = {X 331.5063, Y 25.7713, Z -4.6667, A 0.000, B 0.000, C 0.000 }
gfCNCPoint3[16356] = {X 332.6887, Y 25.4804, Z -4.6667, A 0.000, B 0.000, C 0.000 }
gfCNCPoint3[16357] = {X 333.9031, Y 25.3907, Z -4.6667, A 0.000, B 0.000, C 0.000 }
gfCNCPoint3[16358] = {X 335.1154, Y 25.5046, Z -4.6667, A 0.000, B 0.000, C 0.000 }
gfCNCPoint3[16359] = {X 336.2918, Y 25.8191, Z -4.6667, A 0.000, B 0.000, C 0.000 }
gfCNCPoint3[16360] = {X 337.3993, Y 26.3252, Z -4.6667, A 0.000, B 0.000, C 0.000 }
gfCNCPoint3[16361] = {X 338.1754, Y 26.8291, Z -4.6667, A 0.000, B 0.000, C 0.000 }
gfCNCPoint3[16362] = {X 338.8813, Y 27.4275, Z -4.6667, A 0.000, B 0.000, C 0.000 }
gfCNCPoint3[16363] = {X 339.4535, Y 27.9787, Z -4.6667, A 0.000, B 0.000, C 0.000 }
gfCNCPoint3[16364] = {X 339.8242, Y 28.3633, Z -4.6667, A 0.000, B 0.000, C 0.000 }
gfCNCPoint3[16365] = {X 340.1656, Y 28.7740, Z -4.6667, A 0.000, B 0.000, C 0.000 }
gfCNCPoint3[16366] = {X 345.8671, Y 24.3770, Z -4.6667, A 0.000, B 0.000, C 0.000 }
gfCNCPoint3[16367] = {X 346.4658, Y 25.2131, Z -4.6667, A 0.000, B 0.000, C 0.000 }
gfCNCPoint3[16368] = {X 347.0036, Y 26.0896, Z -4.6667, A 0.000, B 0.000, C 0.000 }
gfCNCPoint3[16369] = {X 347.1062, Y 25.1831, Z -4.6667, A 0.000, B 0.000, C 0.000 }
gfCNCPoint3[16370] = {X 347.1019, Y 24.2708, Z -4.6667, A 0.000, B 0.000, C 0.000 }
gfCNCPoint3[16371] = {X 346.9910, Y 23.3654, Z -4.6667, A 0.000, B 0.000, C 0.000 }
gfCNCPoint3[16372] = {X 346.9495, Y 23.1616, Z -4.6667, A 0.000, B 0.000, C 0.000 }
gfCNCPoint3[16373] = {X 346.8831, Y 22.9646, Z -4.6667, A 0.000, B 0.000, C 0.000 }
gfCNCPoint3[16374] = {X 346.3963, Y 23.6861, Z -4.6667, A 0.000, B 0.000, C 0.000 }
gfCNCPoint3[16375] = {X 345.8671, Y 24.3770, Z -4.6667, A 0.000, B 0.000, C 0.000 }
gfCNCPoint3[16376] = {X 343.9666, Y 25.8427, Z -4.6667, A 0.000, B 0.000, C 0.000 }
gfCNCPoint3[16377] = {X 344.4661, Y 26.5402, Z -4.6667, A 0.000, B 0.000, C 0.000 }
gfCNCPoint3[16378] = {X 344.9147, Y 27.2714, Z -4.6667, A 0.000, B 0.000, C 0.000 }
gfCNCPoint3[16379] = {X 345.4665, Y 28.3745, Z -4.6667, A 0.000, B 0.000, C 0.000 }
gfCNCPoint3[16380] = {X 345.9029, Y 29.5282, Z -4.6667, A 0.000, B 0.000, C 0.000 }
gfCNCPoint3[16381] = {X 346.4603, Y 29.6311, Z -4.6667, A 0.000, B 0.000, C 0.000 }
gfCNCPoint3[16382] = {X 347.0271, Y 29.6221, Z -4.6667, A 0.000, B 0.000, C 0.000 }
gfCNCPoint3[16383] = {X 347.4362, Y 29.5568, Z -4.6667, A 0.000, B 0.000, C 0.000 }
gfCNCPoint3[16384] = {X 347.7945, Y 29.3491, Z -4.6667, A 0.000, B 0.000, C 0.000 }
gfCNCPoint3[16385] = {X 348.4749, Y 28.6294, Z -4.6667, A 0.000, B 0.000, C 0.000 }
gfCNCPoint3[16386] = {X 348.9855, Y 27.7809, Z -4.6667, A 0.000, B 0.000, C 0.000 }
gfCNCPoint3[16387] = {X 349.3028, Y 26.8428, Z -4.6667, A 0.000, B 0.000, C 0.000 }
gfCNCPoint3[16388] = {X 349.3371, Y 26.6710, Z -4.6667, A 0.000, B 0.000, C 0.000 }
gfCNCPoint3[16389] = {X 349.3685, Y 26.4987, Z -4.6667, A 0.000, B 0.000, C 0.000 }
gfCNCPoint3[16390] = {X 349.5020, Y 25.3243, Z -4.6667, A 0.000, B 0.000, C 0.000 }
gfCNCPoint3[16391] = {X 349.4986, Y 24.1425, Z -4.6667, A 0.000, B 0.000, C 0.000 }
gfCNCPoint3[16392] = {X 349.3582, Y 22.9690, Z -4.6667, A 0.000, B 0.000, C 0.000 }
gfCNCPoint3[16393] = {X 349.1802, Y 22.2566, Z -4.6667, A 0.000, B 0.000, C 0.000 }
gfCNCPoint3[16394] = {X 348.8775, Y 21.5877, Z -4.6667, A 0.000, B 0.000, C 0.000 }
gfCNCPoint3[16395] = {X 348.4597, Y 20.9839, Z -4.6667, A 0.000, B 0.000, C 0.000 }
gfCNCPoint3[16396] = {X 348.0927, Y 20.6601, Z -4.6667, A 0.000, B 0.000, C 0.000 }
gfCNCPoint3[16397] = {X 347.6362, Y 20.4836, Z -4.6667, A 0.000, B 0.000, C 0.000 }
gfCNCPoint3[16398] = {X 346.5779, Y 20.3830, Z -4.6667, A 0.000, B 0.000, C 0.000 }
gfCNCPoint3[16399] = {X 345.5197, Y 20.4835, Z -4.6667, A 0.000, B 0.000, C 0.000 }
gfCNCPoint3[16400] = {X 344.7175, Y 21.8940, Z -4.6667, A 0.000, B 0.000, C 0.000 }
gfCNCPoint3[16401] = {X 343.7336, Y 23.1843, Z -4.6667, A 0.000, B 0.000, C 0.000 }
gfCNCPoint3[16402] = {X 342.5857, Y 24.3311, Z -4.6667, A 0.000, B 0.000, C 0.000 }
gfCNCPoint3[16403] = {X 342.7850, Y 24.5231, Z -4.6667, A 0.000, B 0.000, C 0.000 }
gfCNCPoint3[16404] = {X 343.4000, Y 25.1612, Z -4.6667, A 0.000, B 0.000, C 0.000 }
gfCNCPoint3[16405] = {X 343.9666, Y 25.8427, Z -4.6667, A 0.000, B 0.000, C 0.000 }
gfCNCPoint3[16406] = {X 342.0661, Y 27.3083, Z -4.6667, A 0.000, B 0.000, C 0.000 }
gfCNCPoint3[16407] = {X 342.8613, Y 28.5163, Z -4.6667, A 0.000, B 0.000, C 0.000 }
gfCNCPoint3[16408] = {X 343.4676, Y 29.8291, Z -4.6667, A 0.000, B 0.000, C 0.000 }
gfCNCPoint3[16409] = {X 343.8715, Y 31.2177, Z -4.6667, A 0.000, B 0.000, C 0.000 }
gfCNCPoint3[16410] = {X 344.6369, Y 31.6206, Z -4.6667, A 0.000, B 0.000, C 0.000 }
gfCNCPoint3[16411] = {X 345.4580, Y 31.8926, Z -4.6667, A 0.000, B 0.000, C 0.000 }
gfCNCPoint3[16412] = {X 346.3125, Y 32.0264, Z -4.6667, A 0.000, B 0.000, C 0.000 }
gfCNCPoint3[16413] = {X 347.1775, Y 32.0184, Z -4.6667, A 0.000, B 0.000, C 0.000 }
gfCNCPoint3[16414] = {X 347.9595, Y 31.9035, Z -4.6667, A 0.000, B 0.000, C 0.000 }
gfCNCPoint3[16415] = {X 348.6965, Y 31.6178, Z -4.6667, A 0.000, B 0.000, C 0.000 }
gfCNCPoint3[16416] = {X 349.3516, Y 31.1755, Z -4.6667, A 0.000, B 0.000, C 0.000 }
gfCNCPoint3[16417] = {X 350.1528, Y 30.3718, Z -4.6667, A 0.000, B 0.000, C 0.000 }
gfCNCPoint3[16418] = {X 350.8137, Y 29.4493, Z -4.6667, A 0.000, B 0.000, C 0.000 }
gfCNCPoint3[16419] = {X 351.3169, Y 28.4322, Z -4.6667, A 0.000, B 0.000, C 0.000 }
gfCNCPoint3[16420] = {X 351.6493, Y 27.3472, Z -4.6667, A 0.000, B 0.000, C 0.000 }
gfCNCPoint3[16421] = {X 351.8778, Y 25.7621, Z -4.6667, A 0.000, B 0.000, C 0.000 }
gfCNCPoint3[16422] = {X 351.9031, Y 24.1608, Z -4.6667, A 0.000, B 0.000, C 0.000 }
gfCNCPoint3[16423] = {X 351.7248, Y 22.5693, Z -4.6667, A 0.000, B 0.000, C 0.000 }
gfCNCPoint3[16424] = {X 351.4426, Y 21.4555, Z -4.6667, A 0.000, B 0.000, C 0.000 }
gfCNCPoint3[16425] = {X 350.9681, Y 20.4090, Z -4.6667, A 0.000, B 0.000, C 0.000 }
gfCNCPoint3[16426] = {X 350.3162, Y 19.4629, Z -4.6667, A 0.000, B 0.000, C 0.000 }
gfCNCPoint3[16427] = {X 349.6859, Y 18.8473, Z -4.6667, A 0.000, B 0.000, C 0.000 }
gfCNCPoint3[16428] = {X 348.9305, Y 18.3939, Z -4.6667, A 0.000, B 0.000, C 0.000 }
gfCNCPoint3[16429] = {X 348.0908, Y 18.1271, Z -4.6667, A 0.000, B 0.000, C 0.000 }
gfCNCPoint3[16430] = {X 346.9978, Y 17.9941, Z -4.6667, A 0.000, B 0.000, C 0.000 }
gfCNCPoint3[16431] = {X 345.8969, Y 18.0120, Z -4.6667, A 0.000, B 0.000, C 0.000 }
gfCNCPoint3[16432] = {X 344.8088, Y 18.1805, Z -4.6667, A 0.000, B 0.000, C 0.000 }
gfCNCPoint3[16433] = {X 343.7540, Y 18.4964, Z -4.6667, A 0.000, B 0.000, C 0.000 }
gfCNCPoint3[16434] = {X 343.2658, Y 19.6264, Z -4.6667, A 0.000, B 0.000, C 0.000 }
gfCNCPoint3[16435] = {X 342.6383, Y 20.6854, Z -4.6667, A 0.000, B 0.000, C 0.000 }
gfCNCPoint3[16436] = {X 341.8813, Y 21.6562, Z -4.6667, A 0.000, B 0.000, C 0.000 }
gfCNCPoint3[16437] = {X 341.0073, Y 22.5231, Z -4.6667, A 0.000, B 0.000, C 0.000 }
gfCNCPoint3[16438] = {X 340.7217, Y 22.7629, Z -4.6667, A 0.000, B 0.000, C 0.000 }
gfCNCPoint3[16439] = {X 340.4270, Y 22.9916, Z -4.6667, A 0.000, B 0.000, C 0.000 }
gfCNCPoint3[16440] = {X 339.6615, Y 23.5549, Z -4.6667, A 0.000, B 0.000, C 0.000 }
gfCNCPoint3[16441] = {X 339.1299, Y 23.9121, Z -4.6667, A 0.000, B 0.000, C 0.000 }
gfCNCPoint3[16442] = {X 338.5759, Y 24.2333, Z -4.6667, A 0.000, B 0.000, C 0.000 }
gfCNCPoint3[16443] = {X 339.6078, Y 24.9035, Z -4.6667, A 0.000, B 0.000, C 0.000 }
gfCNCPoint3[16444] = {X 340.5464, Y 25.6991, Z -4.6667, A 0.000, B 0.000, C 0.000 }
gfCNCPoint3[16445] = {X 341.1192, Y 26.2509, Z -4.6667, A 0.000, B 0.000, C 0.000 }
gfCNCPoint3[16446] = {X 341.6121, Y 26.7622, Z -4.6667, A 0.000, B 0.000, C 0.000 }
gfCNCPoint3[16447] = {X 342.0661, Y 27.3083, Z -4.6667, A 0.000, B 0.000, C 0.000 }
gfCNCPoint3[16448] = {X 340.1656, Y 28.7740, Z -4.6667, A 0.000, B 0.000, C 0.000 }
gfCNCPoint3[16449] = {X 340.7338, Y 29.6294, Z -4.6667, A 0.000, B 0.000, C 0.000 }
gfCNCPoint3[16450] = {X 341.1760, Y 30.5562, Z -4.6667, A 0.000, B 0.000, C 0.000 }
gfCNCPoint3[16451] = {X 341.4834, Y 31.5360, Z -4.6667, A 0.000, B 0.000, C 0.000 }
gfCNCPoint3[16452] = {X 341.6499, Y 32.5493, Z -4.6667, A 0.000, B 0.000, C 0.000 }
gfCNCPoint3[16453] = {X 341.8460, Y 32.7091, Z -4.6667, A 0.000, B 0.000, C 0.000 }
gfCNCPoint3[16454] = {X 342.0443, Y 32.8663, Z -4.6667, A 0.000, B 0.000, C 0.000 }
gfCNCPoint3[16455] = {X 342.9870, Y 33.4825, Z -4.6667, A 0.000, B 0.000, C 0.000 }
gfCNCPoint3[16456] = {X 344.0099, Y 33.9538, Z -4.6667, A 0.000, B 0.000, C 0.000 }
gfCNCPoint3[16457] = {X 345.0908, Y 34.2702, Z -4.6667, A 0.000, B 0.000, C 0.000 }
gfCNCPoint3[16458] = {X 346.2064, Y 34.4246, Z -4.6667, A 0.000, B 0.000, C 0.000 }
gfCNCPoint3[16459] = {X 347.3326, Y 34.4138, Z -4.6667, A 0.000, B 0.000, C 0.000 }
gfCNCPoint3[16460] = {X 348.3022, Y 34.2883, Z -4.6667, A 0.000, B 0.000, C 0.000 }
gfCNCPoint3[16461] = {X 349.2380, Y 34.0054, Z -4.6667, A 0.000, B 0.000, C 0.000 }
gfCNCPoint3[16462] = {X 350.1146, Y 33.5728, Z -4.6667, A 0.000, B 0.000, C 0.000 }
gfCNCPoint3[16463] = {X 350.9084, Y 33.0020, Z -4.6667, A 0.000, B 0.000, C 0.000 }
gfCNCPoint3[16464] = {X 351.7847, Y 32.1509, Z -4.6667, A 0.000, B 0.000, C 0.000 }
gfCNCPoint3[16465] = {X 352.5434, Y 31.1932, Z -4.6667, A 0.000, B 0.000, C 0.000 }
gfCNCPoint3[16466] = {X 353.1714, Y 30.1453, Z -4.6667, A 0.000, B 0.000, C 0.000 }
gfCNCPoint3[16467] = {X 353.6584, Y 29.0248, Z -4.6667, A 0.000, B 0.000, C 0.000 }
gfCNCPoint3[16468] = {X 353.9959, Y 27.8507, Z -4.6667, A 0.000, B 0.000, C 0.000 }
gfCNCPoint3[16469] = {X 354.2233, Y 26.4400, Z -4.6667, A 0.000, B 0.000, C 0.000 }
gfCNCPoint3[16470] = {X 354.3154, Y 25.0140, Z -4.6667, A 0.000, B 0.000, C 0.000 }
gfCNCPoint3[16471] = {X 354.2712, Y 23.5858, Z -4.6667, A 0.000, B 0.000, C 0.000 }
gfCNCPoint3[16472] = {X 354.0911, Y 22.1683, Z -4.6667, A 0.000, B 0.000, C 0.000 }
gfCNCPoint3[16473] = {X 353.8261, Y 21.0252, Z -4.6667, A 0.000, B 0.000, C 0.000 }
gfCNCPoint3[16474] = {X 353.4127, Y 19.9270, Z -4.6667, A 0.000, B 0.000, C 0.000 }
gfCNCPoint3[16475] = {X 352.8581, Y 18.8929, Z -4.6667, A 0.000, B 0.000, C 0.000 }
gfCNCPoint3[16476] = {X 352.1720, Y 17.9409, Z -4.6667, A 0.000, B 0.000, C 0.000 }
gfCNCPoint3[16477] = {X 351.4221, Y 17.1679, Z -4.6667, A 0.000, B 0.000, C 0.000 }
gfCNCPoint3[16478] = {X 350.5496, Y 16.5366, Z -4.6667, A 0.000, B 0.000, C 0.000 }
gfCNCPoint3[16479] = {X 349.5809, Y 16.0660, Z -4.6667, A 0.000, B 0.000, C 0.000 }
gfCNCPoint3[16480] = {X 348.5452, Y 15.7705, Z -4.6667, A 0.000, B 0.000, C 0.000 }
gfCNCPoint3[16481] = {X 347.1589, Y 15.5993, Z -4.6667, A 0.000, B 0.000, C 0.000 }
gfCNCPoint3[16482] = {X 345.7620, Y 15.6150, Z -4.6667, A 0.000, B 0.000, C 0.000 }
gfCNCPoint3[16483] = {X 344.3799, Y 15.8174, Z -4.6667, A 0.000, B 0.000, C 0.000 }
gfCNCPoint3[16484] = {X 343.0372, Y 16.2028, Z -4.6667, A 0.000, B 0.000, C 0.000 }
gfCNCPoint3[16485] = {X 341.7581, Y 16.7643, Z -4.6667, A 0.000, B 0.000, C 0.000 }
gfCNCPoint3[16486] = {X 341.3706, Y 18.0087, Z -4.6667, A 0.000, B 0.000, C 0.000 }
gfCNCPoint3[16487] = {X 340.7674, Y 19.1641, Z -4.6667, A 0.000, B 0.000, C 0.000 }
gfCNCPoint3[16488] = {X 339.9679, Y 20.1934, Z -4.6667, A 0.000, B 0.000, C 0.000 }
gfCNCPoint3[16489] = {X 338.9976, Y 21.0636, Z -4.6667, A 0.000, B 0.000, C 0.000 }
gfCNCPoint3[16490] = {X 338.2497, Y 21.6141, Z -4.6667, A 0.000, B 0.000, C 0.000 }
gfCNCPoint3[16491] = {X 337.8538, Y 21.8795, Z -4.6667, A 0.000, B 0.000, C 0.000 }
gfCNCPoint3[16492] = {X 337.4413, Y 22.1185, Z -4.6667, A 0.000, B 0.000, C 0.000 }
gfCNCPoint3[16493] = {X 336.3239, Y 22.6023, Z -4.6667, A 0.000, B 0.000, C 0.000 }
gfCNCPoint3[16494] = {X 335.1415, Y 22.8932, Z -4.6667, A 0.000, B 0.000, C 0.000 }
gfCNCPoint3[16495] = {X 333.9271, Y 22.9829, Z -4.6667, A 0.000, B 0.000, C 0.000 }
gfCNCPoint3[16496] = {X 332.7148, Y 22.8690, Z -4.6667, A 0.000, B 0.000, C 0.000 }
gfCNCPoint3[16497] = {X 331.5384, Y 22.5546, Z -4.6667, A 0.000, B 0.000, C 0.000 }
gfCNCPoint3[16498] = {X 330.4309, Y 22.0485, Z -4.6667, A 0.000, B 0.000, C 0.000 }
gfCNCPoint3[16499] = {X 329.5144, Y 21.4374, Z -4.6667, A 0.000, B 0.000, C 0.000 }
gfCNCPoint3[16500] = {X 328.7005, Y 20.6950, Z -4.6667, A 0.000, B 0.000, C 0.000 }
gfCNCPoint3[16501] = {X 328.0081, Y 19.8382, Z -4.6667, A 0.000, B 0.000, C 0.000 }
gfCNCPoint3[16502] = {X 327.4528, Y 18.8869, Z -4.6667, A 0.000, B 0.000, C 0.000 }
gfCNCPoint3[16503] = {X 323.9321, Y 11.6443, Z -4.6667, A 0.000, B 0.000, C 0.000 }
gfCNCPoint3[16504] = {X 323.5337, Y 10.6421, Z -4.6667, A 0.000, B 0.000, C 0.000 }
gfCNCPoint3[16505] = {X 323.2878, Y 9.5921, Z -4.6667, A 0.000, B 0.000, C 0.000 }
gfCNCPoint3[16506] = {X 323.1997, Y 8.5173, Z -4.6667, A 0.000, B 0.000, C 0.000 }
gfCNCPoint3[16507] = {X 323.2713, Y 7.4413, Z -4.6667, A 0.000, B 0.000, C 0.000 }
gfCNCPoint3[16508] = {X 323.4720, Y 6.4884, Z -4.6667, A 0.000, B 0.000, C 0.000 }
gfCNCPoint3[16509] = {X 323.7980, Y 5.5708, Z -4.6667, A 0.000, B 0.000, C 0.000 }
gfCNCPoint3[16510] = {X 324.2436, Y 4.7050, Z -4.6667, A 0.000, B 0.000, C 0.000 }
gfCNCPoint3[16511] = {X 168.0206, Y 4.7050, Z -4.6667, A 0.000, B 0.000, C 0.000 }
gfCNCPoint3[16512] = {X 168.0206, Y 9.5050, Z -4.6667, A 0.000, B 0.000, C 0.000 }
gfCNCPoint3[16513] = {X 166.5360, Y 9.5050, Z -4.6667, A 0.000, B 0.000, C 0.000 }
gfCNCPoint3[16514] = {X 166.5855, Y 9.9931, Z -4.6667, A 0.000, B 0.000, C 0.000 }
gfCNCPoint3[16515] = {X 166.6021, Y 10.4835, Z -4.6667, A 0.000, B 0.000, C 0.000 }
gfCNCPoint3[16516] = {X 166.6021, Y 13.0969, Z -4.6667, A 0.000, B 0.000, C 0.000 }
gfCNCPoint3[16517] = {X 166.8569, Y 11.8210, Z -4.6667, A 0.000, B 0.000, C 0.000 }
gfCNCPoint3[16518] = {X 167.3348, Y 10.6108, Z -4.6667, A 0.000, B 0.000, C 0.000 }
gfCNCPoint3[16519] = {X 168.0206, Y 9.5050, Z -4.6667, A 0.000, B 0.000, C 0.000 }
gfCNCPoint3[16520] = {X 168.0206, Y 7.1050, Z -4.6667, A 0.000, B 0.000, C 0.000 }
gfCNCPoint3[16521] = {X 162.8434, Y 7.1050, Z -4.6667, A 0.000, B 0.000, C 0.000 }
gfCNCPoint3[16522] = {X 163.4703, Y 7.9131, Z -4.6667, A 0.000, B 0.000, C 0.000 }
gfCNCPoint3[16523] = {X 163.9149, Y 8.8341, Z -4.6667, A 0.000, B 0.000, C 0.000 }
gfCNCPoint3[16524] = {X 164.1578, Y 9.8276, Z -4.6667, A 0.000, B 0.000, C 0.000 }
gfCNCPoint3[16525] = {X 164.1910, Y 10.1548, Z -4.6667, A 0.000, B 0.000, C 0.000 }
gfCNCPoint3[16526] = {X 164.2021, Y 10.4835, Z -4.6667, A 0.000, B 0.000, C 0.000 }
gfCNCPoint3[16527] = {X 164.2021, Y 17.4615, Z -4.6667, A 0.000, B 0.000, C 0.000 }
gfCNCPoint3[16528] = {X 164.1139, Y 18.3848, Z -4.6667, A 0.000, B 0.000, C 0.000 }
gfCNCPoint3[16529] = {X 163.8527, Y 19.2748, Z -4.6667, A 0.000, B 0.000, C 0.000 }
gfCNCPoint3[16530] = {X 163.4278, Y 20.0992, Z -4.6667, A 0.000, B 0.000, C 0.000 }
gfCNCPoint3[16531] = {X 162.8546, Y 20.8283, Z -4.6667, A 0.000, B 0.000, C 0.000 }
gfCNCPoint3[16532] = {X 162.1539, Y 21.4359, Z -4.6667, A 0.000, B 0.000, C 0.000 }
gfCNCPoint3[16533] = {X 161.3508, Y 21.8999, Z -4.6667, A 0.000, B 0.000, C 0.000 }
gfCNCPoint3[16534] = {X 160.4744, Y 22.2035, Z -4.6667, A 0.000, B 0.000, C 0.000 }
gfCNCPoint3[16535] = {X 162.1746, Y 29.1999, Z -4.6667, A 0.000, B 0.000, C 0.000 }
gfCNCPoint3[16536] = {X 161.1124, Y 29.4081, Z -4.6667, A 0.000, B 0.000, C 0.000 }
gfCNCPoint3[16537] = {X 160.0358, Y 29.5204, Z -4.6667, A 0.000, B 0.000, C 0.000 }
gfCNCPoint3[16538] = {X 160.0353, Y 38.3364, Z -4.6667, A 0.000, B 0.000, C 0.000 }
gfCNCPoint3[16539] = {X 160.6835, Y 39.6936, Z -4.6667, A 0.000, B 0.000, C 0.000 }
gfCNCPoint3[16540] = {X 161.1585, Y 41.1206, Z -4.6667, A 0.000, B 0.000, C 0.000 }
gfCNCPoint3[16541] = {X 162.0478, Y 41.1205, Z -4.6667, A 0.000, B 0.000, C 0.000 }
gfCNCPoint3[16542] = {X 161.6734, Y 39.3707, Z -4.6667, A 0.000, B 0.000, C 0.000 }
gfCNCPoint3[16543] = {X 161.4494, Y 37.5955, Z -4.6667, A 0.000, B 0.000, C 0.000 }
gfCNCPoint3[16544] = {X 161.3314, Y 35.4802, Z -4.6667, A 0.000, B 0.000, C 0.000 }
gfCNCPoint3[16545] = {X 161.4136, Y 33.3633, Z -4.6667, A 0.000, B 0.000, C 0.000 }
gfCNCPoint3[16546] = {X 161.6956, Y 31.2636, Z -4.6667, A 0.000, B 0.000, C 0.000 }
gfCNCPoint3[16547] = {X 162.1746, Y 29.1999, Z -4.6667, A 0.000, B 0.000, C 0.000 }
gfCNCPoint3[16548] = {X 161.6079, Y 26.8678, Z -4.6667, A 0.000, B 0.000, C 0.000 }
gfCNCPoint3[16549] = {X 160.4731, Y 27.0729, Z -4.6667, A 0.000, B 0.000, C 0.000 }
gfCNCPoint3[16550] = {X 159.3220, Y 27.1415, Z -4.6667, A 0.000, B 0.000, C 0.000 }
gfCNCPoint3[16551] = {X 158.6569, Y 27.1415, Z -4.6667, A 0.000, B 0.000, C 0.000 }
gfCNCPoint3[16552] = {X 158.1457, Y 27.1259, Z -4.6667, A 0.000, B 0.000, C 0.000 }
gfCNCPoint3[16553] = {X 157.6360, Y 27.0834, Z -4.6667, A 0.000, B 0.000, C 0.000 }
gfCNCPoint3[16554] = {X 157.6352, Y 38.9960, Z -4.6667, A 0.000, B 0.000, C 0.000 }
gfCNCPoint3[16555] = {X 158.2191, Y 40.0483, Z -4.6667, A 0.000, B 0.000, C 0.000 }
gfCNCPoint3[16556] = {X 158.6683, Y 41.1648, Z -4.6667, A 0.000, B 0.000, C 0.000 }
gfCNCPoint3[16557] = {X 158.9761, Y 42.3283, Z -4.6667, A 0.000, B 0.000, C 0.000 }
gfCNCPoint3[16558] = {X 159.1375, Y 43.5209, Z -4.6667, A 0.000, B 0.000, C 0.000 }
gfCNCPoint3[16559] = {X 165.4296, Y 43.5200, Z -4.6667, A 0.000, B 0.000, C 0.000 }
gfCNCPoint3[16560] = {X 164.8361, Y 42.0421, Z -4.6667, A 0.000, B 0.000, C 0.000 }
gfCNCPoint3[16561] = {X 164.3712, Y 40.5188, Z -4.6667, A 0.000, B 0.000, C 0.000 }
gfCNCPoint3[16562] = {X 164.0376, Y 38.9572, Z -4.6667, A 0.000, B 0.000, C 0.000 }
gfCNCPoint3[16563] = {X 163.8392, Y 37.3727, Z -4.6667, A 0.000, B 0.000, C 0.000 }
gfCNCPoint3[16564] = {X 163.7314, Y 35.4781, Z -4.6667, A 0.000, B 0.000, C 0.000 }
gfCNCPoint3[16565] = {X 163.8037, Y 33.5819, Z -4.6667, A 0.000, B 0.000, C 0.000 }
gfCNCPoint3[16566] = {X 164.0554, Y 31.7011, Z -4.6667, A 0.000, B 0.000, C 0.000 }
gfCNCPoint3[16567] = {X 164.4841, Y 29.8525, Z -4.6667, A 0.000, B 0.000, C 0.000 }
gfCNCPoint3[16568] = {X 164.8362, Y 28.7331, Z -4.6667, A 0.000, B 0.000, C 0.000 }
gfCNCPoint3[16569] = {X 165.2534, Y 27.6363, Z -4.6667, A 0.000, B 0.000, C 0.000 }
gfCNCPoint3[16570] = {X 165.8699, Y 26.3055, Z -4.6667, A 0.000, B 0.000, C 0.000 }
gfCNCPoint3[16571] = {X 166.6042, Y 25.0358, Z -4.6667, A 0.000, B 0.000, C 0.000 }
gfCNCPoint3[16572] = {X 167.4502, Y 23.8377, Z -4.6667, A 0.000, B 0.000, C 0.000 }
gfCNCPoint3[16573] = {X 167.1640, Y 23.1367, Z -4.6667, A 0.000, B 0.000, C 0.000 }
gfCNCPoint3[16574] = {X 166.2873, Y 24.1837, Z -4.6667, A 0.000, B 0.000, C 0.000 }
gfCNCPoint3[16575] = {X 165.2720, Y 25.0970, Z -4.6667, A 0.000, B 0.000, C 0.000 }
gfCNCPoint3[16576] = {X 164.1383, Y 25.8583, Z -4.6667, A 0.000, B 0.000, C 0.000 }
gfCNCPoint3[16577] = {X 162.9088, Y 26.4525, Z -4.6667, A 0.000, B 0.000, C 0.000 }
gfCNCPoint3[16578] = {X 161.6079, Y 26.8678, Z -4.6667, A 0.000, B 0.000, C 0.000 }
gfCNCPoint3[16579] = {X 161.0411, Y 24.5357, Z -4.6667, A 0.000, B 0.000, C 0.000 }
gfCNCPoint3[16580] = {X 160.1877, Y 24.6899, Z -4.6667, A 0.000, B 0.000, C 0.000 }
gfCNCPoint3[16581] = {X 159.3220, Y 24.7415, Z -4.6667, A 0.000, B 0.000, C 0.000 }
gfCNCPoint3[16582] = {X 158.6669, Y 24.7415, Z -4.6667, A 0.000, B 0.000, C 0.000 }
gfCNCPoint3[16583] = {X 158.2820, Y 24.7298, Z -4.6667, A 0.000, B 0.000, C 0.000 }
gfCNCPoint3[16584] = {X 157.8982, Y 24.6978, Z -4.6667, A 0.000, B 0.000, C 0.000 }
gfCNCPoint3[16585] = {X 156.9780, Y 24.5366, Z -4.6667, A 0.000, B 0.000, C 0.000 }
gfCNCPoint3[16586] = {X 156.0858, Y 24.2595, Z -4.6667, A 0.000, B 0.000, C 0.000 }
gfCNCPoint3[16587] = {X 155.2362, Y 23.8708, Z -4.6667, A 0.000, B 0.000, C 0.000 }
gfCNCPoint3[16588] = {X 155.2352, Y 39.7518, Z -4.6667, A 0.000, B 0.000, C 0.000 }
gfCNCPoint3[16589] = {X 155.8259, Y 40.6436, Z -4.6667, A 0.000, B 0.000, C 0.000 }
gfCNCPoint3[16590] = {X 156.2803, Y 41.6121, Z -4.6667, A 0.000, B 0.000, C 0.000 }
gfCNCPoint3[16591] = {X 156.5884, Y 42.6366, Z -4.6667, A 0.000, B 0.000, C 0.000 }
gfCNCPoint3[16592] = {X 156.7439, Y 43.6950, Z -4.6667, A 0.000, B 0.000, C 0.000 }
gfCNCPoint3[16593] = {X 156.7579, Y 43.9477, Z -4.6667, A 0.000, B 0.000, C 0.000 }
gfCNCPoint3[16594] = {X 156.7631, Y 44.2008, Z -4.6667, A 0.000, B 0.000, C 0.000 }
gfCNCPoint3[16595] = {X 156.7629, Y 45.0587, Z -4.6667, A 0.000, B 0.000, C 0.000 }
gfCNCPoint3[16596] = {X 156.7352, Y 45.6370, Z -4.6667, A 0.000, B 0.000, C 0.000 }
gfCNCPoint3[16597] = {X 156.6616, Y 46.2112, Z -4.6667, A 0.000, B 0.000, C 0.000 }
gfCNCPoint3[16598] = {X 157.9053, Y 46.0005, Z -4.6667, A 0.000, B 0.000, C 0.000 }
gfCNCPoint3[16599] = {X 159.1641, Y 45.9207, Z -4.6667, A 0.000, B 0.000, C 0.000 }
gfCNCPoint3[16600] = {X 159.2310, Y 45.9202, Z -4.6667, A 0.000, B 0.000, C 0.000 }
gfCNCPoint3[16601] = {X 159.2980, Y 45.9200, Z -4.6667, A 0.000, B 0.000, C 0.000 }
gfCNCPoint3[16602] = {X 169.6829, Y 45.9200, Z -4.6667, A 0.000, B 0.000, C 0.000 }
gfCNCPoint3[16603] = {X 168.9022, Y 44.8481, Z -4.6667, A 0.000, B 0.000, C 0.000 }
gfCNCPoint3[16604] = {X 168.2118, Y 43.7159, Z -4.6667, A 0.000, B 0.000, C 0.000 }
gfCNCPoint3[16605] = {X 167.6164, Y 42.5310, Z -4.6667, A 0.000, B 0.000, C 0.000 }
gfCNCPoint3[16606] = {X 166.9483, Y 40.7946, Z -4.6667, A 0.000, B 0.000, C 0.000 }
gfCNCPoint3[16607] = {X 166.4838, Y 38.9930, Z -4.6667, A 0.000, B 0.000, C 0.000 }
gfCNCPoint3[16608] = {X 166.2290, Y 37.1500, Z -4.6667, A 0.000, B 0.000, C 0.000 }
gfCNCPoint3[16609] = {X 166.1309, Y 35.3975, Z -4.6667, A 0.000, B 0.000, C 0.000 }
gfCNCPoint3[16610] = {X 166.2078, Y 33.6439, Z -4.6667, A 0.000, B 0.000, C 0.000 }
gfCNCPoint3[16611] = {X 166.4590, Y 31.9067, Z -4.6667, A 0.000, B 0.000, C 0.000 }
gfCNCPoint3[16612] = {X 166.8820, Y 30.2032, Z -4.6667, A 0.000, B 0.000, C 0.000 }
gfCNCPoint3[16613] = {X 167.4726, Y 28.5502, Z -4.6667, A 0.000, B 0.000, C 0.000 }
gfCNCPoint3[16614] = {X 168.2333, Y 26.9811, Z -4.6667, A 0.000, B 0.000, C 0.000 }
gfCNCPoint3[16615] = {X 169.1856, Y 25.5202, Z -4.6667, A 0.000, B 0.000, C 0.000 }
gfCNCPoint3[16616] = {X 170.3142, Y 24.1909, Z -4.6667, A 0.000, B 0.000, C 0.000 }
gfCNCPoint3[16617] = {X 169.9865, Y 23.6222, Z -4.6667, A 0.000, B 0.000, C 0.000 }
gfCNCPoint3[16618] = {X 169.7112, Y 23.0264, Z -4.6667, A 0.000, B 0.000, C 0.000 }
gfCNCPoint3[16619] = {X 167.1001, Y 16.6309, Z -4.6667, A 0.000, B 0.000, C 0.000 }
gfCNCPoint3[16620] = {X 166.7820, Y 15.6636, Z -4.6667, A 0.000, B 0.000, C 0.000 }
gfCNCPoint3[16621] = {X 166.6021, Y 14.6613, Z -4.6667, A 0.000, B 0.000, C 0.000 }
gfCNCPoint3[16622] = {X 166.6021, Y 17.4615, Z -4.6667, A 0.000, B 0.000, C 0.000 }
gfCNCPoint3[16623] = {X 166.5130, Y 18.5970, Z -4.6667, A 0.000, B 0.000, C 0.000 }
gfCNCPoint3[16624] = {X 166.2479, Y 19.7047, Z -4.6667, A 0.000, B 0.000, C 0.000 }
gfCNCPoint3[16625] = {X 165.8132, Y 20.7575, Z -4.6667, A 0.000, B 0.000, C 0.000 }
gfCNCPoint3[16626] = {X 165.2197, Y 21.7296, Z -4.6667, A 0.000, B 0.000, C 0.000 }
gfCNCPoint3[16627] = {X 164.3787, Y 22.6988, Z -4.6667, A 0.000, B 0.000, C 0.000 }
gfCNCPoint3[16628] = {X 163.3806, Y 23.5053, Z -4.6667, A 0.000, B 0.000, C 0.000 }
gfCNCPoint3[16629] = {X 162.2565, Y 24.1240, Z -4.6667, A 0.000, B 0.000, C 0.000 }
gfCNCPoint3[16630] = {X 161.0411, Y 24.5357, Z -4.6667, A 0.000, B 0.000, C 0.000 }
gfCNCPoint3[16631] = {X 160.4744, Y 22.2035, Z -4.6667, A 0.000, B 0.000, C 0.000 }
gfCNCPoint3[16632] = {X 159.9023, Y 22.3069, Z -4.6667, A 0.000, B 0.000, C 0.000 }
gfCNCPoint3[16633] = {X 159.3220, Y 22.3415, Z -4.6667, A 0.000, B 0.000, C 0.000 }
gfCNCPoint3[16634] = {X 158.6769, Y 22.3415, Z -4.6667, A 0.000, B 0.000, C 0.000 }
gfCNCPoint3[16635] = {X 157.8801, Y 22.2731, Z -4.6667, A 0.000, B 0.000, C 0.000 }
gfCNCPoint3[16636] = {X 157.1049, Y 22.0764, Z -4.6667, A 0.000, B 0.000, C 0.000 }
gfCNCPoint3[16637] = {X 156.3719, Y 21.7565, Z -4.6667, A 0.000, B 0.000, C 0.000 }
gfCNCPoint3[16638] = {X 155.5229, Y 21.1787, Z -4.6667, A 0.000, B 0.000, C 0.000 }
gfCNCPoint3[16639] = {X 154.8125, Y 20.4371, Z -4.6667, A 0.000, B 0.000, C 0.000 }
gfCNCPoint3[16640] = {X 152.8364, Y 20.4379, Z -4.6667, A 0.000, B 0.000, C 0.000 }
gfCNCPoint3[16641] = {X 152.8351, Y 40.6542, Z -4.6667, A 0.000, B 0.000, C 0.000 }
gfCNCPoint3[16642] = {X 153.1751, Y 41.0219, Z -4.6667, A 0.000, B 0.000, C 0.000 }
gfCNCPoint3[16643] = {X 153.6798, Y 41.7260, Z -4.6667, A 0.000, B 0.000, C 0.000 }
gfCNCPoint3[16644] = {X 154.0531, Y 42.5077, Z -4.6667, A 0.000, B 0.000, C 0.000 }
gfCNCPoint3[16645] = {X 154.2832, Y 43.3428, Z -4.6667, A 0.000, B 0.000, C 0.000 }
gfCNCPoint3[16646] = {X 154.3631, Y 44.2054, Z -4.6667, A 0.000, B 0.000, C 0.000 }
gfCNCPoint3[16647] = {X 154.3629, Y 45.0469, Z -4.6667, A 0.000, B 0.000, C 0.000 }
gfCNCPoint3[16648] = {X 154.3441, Y 45.4307, Z -4.6667, A 0.000, B 0.000, C 0.000 }
gfCNCPoint3[16649] = {X 154.2951, Y 45.8119, Z -4.6667, A 0.000, B 0.000, C 0.000 }
gfCNCPoint3[16650] = {X 154.0370, Y 46.7541, Z -4.6667, A 0.000, B 0.000, C 0.000 }
gfCNCPoint3[16651] = {X 153.5963, Y 47.6260, Z -4.6667, A 0.000, B 0.000, C 0.000 }
gfCNCPoint3[16652] = {X 152.9909, Y 48.3926, Z -4.6667, A 0.000, B 0.000, C 0.000 }
gfCNCPoint3[16653] = {X 152.2448, Y 49.0233, Z -4.6667, A 0.000, B 0.000, C 0.000 }
gfCNCPoint3[16654] = {X 151.3881, Y 49.4928, Z -4.6667, A 0.000, B 0.000, C 0.000 }
gfCNCPoint3[16655] = {X 150.4551, Y 49.7822, Z -4.6667, A 0.000, B 0.000, C 0.000 }
gfCNCPoint3[16656] = {X 149.4831, Y 49.8800, Z -4.6667, A 0.000, B 0.000, C 0.000 }
gfCNCPoint3[16657] = {X 143.0396, Y 49.8800, Z -4.6667, A 0.000, B 0.000, C 0.000 }
gfCNCPoint3[16658] = {X 142.0923, Y 49.7872, Z -4.6667, A 0.000, B 0.000, C 0.000 }
gfCNCPoint3[16659] = {X 141.1811, Y 49.5122, Z -4.6667, A 0.000, B 0.000, C 0.000 }
gfCNCPoint3[16660] = {X 140.3405, Y 49.0656, Z -4.6667, A 0.000, B 0.000, C 0.000 }
gfCNCPoint3[16661] = {X 139.6026, Y 48.4643, Z -4.6667, A 0.000, B 0.000, C 0.000 }
gfCNCPoint3[16662] = {X 138.9955, Y 47.7312, Z -4.6667, A 0.000, B 0.000, C 0.000 }
gfCNCPoint3[16663] = {X 138.5423, Y 46.8942, Z -4.6667, A 0.000, B 0.000, C 0.000 }
gfCNCPoint3[16664] = {X 138.2601, Y 45.9852, Z -4.6667, A 0.000, B 0.000, C 0.000 }
gfCNCPoint3[16665] = {X 138.1598, Y 45.0386, Z -4.6667, A 0.000, B 0.000, C 0.000 }
gfCNCPoint3[16666] = {X 138.1601, Y 44.1416, Z -4.6667, A 0.000, B 0.000, C 0.000 }
gfCNCPoint3[16667] = {X 138.2148, Y 43.4769, Z -4.6667, A 0.000, B 0.000, C 0.000 }
gfCNCPoint3[16668] = {X 138.3597, Y 42.8258, Z -4.6667, A 0.000, B 0.000, C 0.000 }
gfCNCPoint3[16669] = {X 129.1532, Y 40.1052, Z -4.6667, A 0.000, B 0.000, C 0.000 }
gfCNCPoint3[16670] = {X 129.5665, Y 38.9035, Z -4.6667, A 0.000, B 0.000, C 0.000 }
gfCNCPoint3[16671] = {X 130.0836, Y 37.7426, Z -4.6667, A 0.000, B 0.000, C 0.000 }
gfCNCPoint3[16672] = {X 130.0836, Y 31.6021, Z -4.6667, A 0.000, B 0.000, C 0.000 }
gfCNCPoint3[16673] = {X 129.2062, Y 31.3797, Z -4.6667, A 0.000, B 0.000, C 0.000 }
gfCNCPoint3[16674] = {X 128.3445, Y 31.1030, Z -4.6667, A 0.000, B 0.000, C 0.000 }
gfCNCPoint3[16675] = {X 128.3442, Y 38.3292, Z -4.6667, A 0.000, B 0.000, C 0.000 }
gfCNCPoint3[16676] = {X 128.7846, Y 39.2009, Z -4.6667, A 0.000, B 0.000, C 0.000 }
gfCNCPoint3[16677] = {X 129.1532, Y 40.1052, Z -4.6667, A 0.000, B 0.000, C 0.000 }
gfCNCPoint3[16678] = {X 131.4548, Y 40.7854, Z -4.6667, A 0.000, B 0.000, C 0.000 }
gfCNCPoint3[16679] = {X 131.9017, Y 39.5320, Z -4.6667, A 0.000, B 0.000, C 0.000 }
gfCNCPoint3[16680] = {X 132.4836, Y 38.3354, Z -4.6667, A 0.000, B 0.000, C 0.000 }
gfCNCPoint3[16681] = {X 132.4836, Y 29.5202, Z -4.6667, A 0.000, B 0.000, C 0.000 }
gfCNCPoint3[16682] = {X 131.3525, Y 29.3993, Z -4.6667, A 0.000, B 0.000, C 0.000 }
gfCNCPoint3[16683] = {X 130.2378, Y 29.1726, Z -4.6667, A 0.000, B 0.000, C 0.000 }
gfCNCPoint3[16684] = {X 129.1494, Y 28.8419, Z -4.6667, A 0.000, B 0.000, C 0.000 }
gfCNCPoint3[16685] = {X 128.0250, Y 28.3766, Z -4.6667, A 0.000, B 0.000, C 0.000 }
gfCNCPoint3[16686] = {X 126.9531, Y 27.8005, Z -4.6667, A 0.000, B 0.000, C 0.000 }
gfCNCPoint3[16687] = {X 125.9447, Y 27.1195, Z -4.6667, A 0.000, B 0.000, C 0.000 }
gfCNCPoint3[16688] = {X 125.9441, Y 38.9898, Z -4.6667, A 0.000, B 0.000, C 0.000 }
gfCNCPoint3[16689] = {X 126.4739, Y 39.9286, Z -4.6667, A 0.000, B 0.000, C 0.000 }
gfCNCPoint3[16690] = {X 126.8960, Y 40.9205, Z -4.6667, A 0.000, B 0.000, C 0.000 }
gfCNCPoint3[16691] = {X 127.2098, Y 41.9730, Z -4.6667, A 0.000, B 0.000, C 0.000 }
gfCNCPoint3[16692] = {X 127.4025, Y 43.0542, Z -4.6667, A 0.000, B 0.000, C 0.000 }
gfCNCPoint3[16693] = {X 127.4714, Y 44.1502, Z -4.6667, A 0.000, B 0.000, C 0.000 }
gfCNCPoint3[16694] = {X 127.4716, Y 45.0000, Z -4.6667, A 0.000, B 0.000, C 0.000 }
gfCNCPoint3[16695] = {X 127.4070, Y 46.1159, Z -4.6667, A 0.000, B 0.000, C 0.000 }
gfCNCPoint3[16696] = {X 127.2143, Y 47.2168, Z -4.6667, A 0.000, B 0.000, C 0.000 }
gfCNCPoint3[16697] = {X 126.8960, Y 48.2883, Z -4.6667, A 0.000, B 0.000, C 0.000 }
gfCNCPoint3[16698] = {X 126.2883, Y 49.6376, Z -4.6667, A 0.000, B 0.000, C 0.000 }
gfCNCPoint3[16699] = {X 125.4821, Y 50.8786, Z -4.6667, A 0.000, B 0.000, C 0.000 }
gfCNCPoint3[16700] = {X 124.4962, Y 51.9821, Z -4.6667, A 0.000, B 0.000, C 0.000 }
gfCNCPoint3[16701] = {X 123.3536, Y 52.9225, Z -4.6667, A 0.000, B 0.000, C 0.000 }
gfCNCPoint3[16702] = {X 122.0810, Y 53.6778, Z -4.6667, A 0.000, B 0.000, C 0.000 }
gfCNCPoint3[16703] = {X 120.7081, Y 54.2302, Z -4.6667, A 0.000, B 0.000, C 0.000 }
gfCNCPoint3[16704] = {X 119.2671, Y 54.5669, Z -4.6667, A 0.000, B 0.000, C 0.000 }
gfCNCPoint3[16705] = {X 117.7916, Y 54.6800, Z -4.6667, A 0.000, B 0.000, C 0.000 }
gfCNCPoint3[16706] = {X 111.9185, Y 54.6800, Z -4.6667, A 0.000, B 0.000, C 0.000 }
gfCNCPoint3[16707] = {X 111.7456, Y 54.6785, Z -4.6667, A 0.000, B 0.000, C 0.000 }
gfCNCPoint3[16708] = {X 111.5728, Y 54.6738, Z -4.6667, A 0.000, B 0.000, C 0.000 }
gfCNCPoint3[16709] = {X 111.0585, Y 69.0646, Z -4.6667, A 0.000, B 0.000, C 0.000 }
gfCNCPoint3[16710] = {X 109.0296, Y 68.9061, Z -4.6667, A 0.000, B 0.000, C 0.000 }
gfCNCPoint3[16711] = {X 107.0213, Y 68.5768, Z -4.6667, A 0.000, B 0.000, C 0.000 }
gfCNCPoint3[16712] = {X 105.0765, Y 68.8983, Z -4.6667, A 0.000, B 0.000, C 0.000 }
gfCNCPoint3[16713] = {X 103.1119, Y 69.0597, Z -4.6667, A 0.000, B 0.000, C 0.000 }
gfCNCPoint3[16714] = {X 101.1407, Y 69.0599, Z -4.6667, A 0.000, B 0.000, C 0.000 }
gfCNCPoint3[16715] = {X 99.1761, Y 68.8989, Z -4.6667, A 0.000, B 0.000, C 0.000 }
gfCNCPoint3[16716] = {X 97.2313, Y 68.5777, Z -4.6667, A 0.000, B 0.000, C 0.000 }
gfCNCPoint3[16717] = {X 95.6131, Y 68.8563, Z -4.6667, A 0.000, B 0.000, C 0.000 }
gfCNCPoint3[16718] = {X 93.9796, Y 69.0240, Z -4.6667, A 0.000, B 0.000, C 0.000 }
gfCNCPoint3[16719] = {X 92.3385, Y 69.0800, Z -4.6667, A 0.000, B 0.000, C 0.000 }
gfCNCPoint3[16720] = {X 86.6884, Y 69.0800, Z -4.6667, A 0.000, B 0.000, C 0.000 }
gfCNCPoint3[16721] = {X 84.7316, Y 70.2668, Z -4.6667, A 0.000, B 0.000, C 0.000 }
gfCNCPoint3[16722] = {X 82.6871, Y 71.2950, Z -4.6667, A 0.000, B 0.000, C 0.000 }
gfCNCPoint3[16723] = {X 107.2715, Y 71.2950, Z -4.6667, A 0.000, B 0.000, C 0.000 }
gfCNCPoint3[16724] = {X 109.1258, Y 70.1132, Z -4.6667, A 0.000, B 0.000, C 0.000 }
gfCNCPoint3[16725] = {X 111.0585, Y 69.0646, Z -4.6667, A 0.000, B 0.000, C 0.000 }
gfCNCPoint3[16726] = {X 111.1442, Y 66.6662, Z -4.6667, A 0.000, B 0.000, C 0.000 }
gfCNCPoint3[16727] = {X 109.0696, Y 66.4920, Z -4.6667, A 0.000, B 0.000, C 0.000 }
gfCNCPoint3[16728] = {X 107.0213, Y 66.1197, Z -4.6667, A 0.000, B 0.000, C 0.000 }
gfCNCPoint3[16729] = {X 105.0796, Y 66.4776, Z -4.6667, A 0.000, B 0.000, C 0.000 }
gfCNCPoint3[16730] = {X 103.1135, Y 66.6574, Z -4.6667, A 0.000, B 0.000, C 0.000 }
gfCNCPoint3[16731] = {X 101.1392, Y 66.6576, Z -4.6667, A 0.000, B 0.000, C 0.000 }
gfCNCPoint3[16732] = {X 99.1730, Y 66.4782, Z -4.6667, A 0.000, B 0.000, C 0.000 }
gfCNCPoint3[16733] = {X 97.2313, Y 66.1207, Z -4.6667, A 0.000, B 0.000, C 0.000 }
gfCNCPoint3[16734] = {X 95.6161, Y 66.4308, Z -4.6667, A 0.000, B 0.000, C 0.000 }
gfCNCPoint3[16735] = {X 93.9821, Y 66.6176, Z -4.6667, A 0.000, B 0.000, C 0.000 }
gfCNCPoint3[16736] = {X 92.3385, Y 66.6800, Z -4.6667, A 0.000, B 0.000, C 0.000 }
gfCNCPoint3[16737] = {X 85.9487, Y 66.6800, Z -4.6667, A 0.000, B 0.000, C 0.000 }
gfCNCPoint3[16738] = {X 83.8779, Y 67.9935, Z -4.6667, A 0.000, B 0.000, C 0.000 }
gfCNCPoint3[16739] = {X 81.6946, Y 69.1098, Z -4.6667, A 0.000, B 0.000, C 0.000 }
gfCNCPoint3[16740] = {X 79.6016, Y 69.9548, Z -4.6667, A 0.000, B 0.000, C 0.000 }
gfCNCPoint3[16741] = {X 77.4442, Y 70.6184, Z -4.6667, A 0.000, B 0.000, C 0.000 }
gfCNCPoint3[16742] = {X 75.2382, Y 71.0959, Z -4.6667, A 0.000, B 0.000, C 0.000 }
gfCNCPoint3[16743] = {X 72.9995, Y 71.3838, Z -4.6667, A 0.000, B 0.000, C 0.000 }
gfCNCPoint3[16744] = {X 70.7445, Y 71.4800, Z -4.6667, A 0.000, B 0.000, C 0.000 }
gfCNCPoint3[16745] = {X 64.1851, Y 71.4800, Z -4.6667, A 0.000, B 0.000, C 0.000 }
gfCNCPoint3[16746] = {X 62.0752, Y 71.3958, Z -4.6667, A 0.000, B 0.000, C 0.000 }
gfCNCPoint3[16747] = {X 59.9787, Y 71.1438, Z -4.6667, A 0.000, B 0.000, C 0.000 }
gfCNCPoint3[16748] = {X 57.9089, Y 70.7255, Z -4.6667, A 0.000, B 0.000, C 0.000 }
gfCNCPoint3[16749] = {X 55.8790, Y 70.1436, Z -4.6667, A 0.000, B 0.000, C 0.000 }
gfCNCPoint3[16750] = {X 53.8492, Y 70.7255, Z -4.6667, A 0.000, B 0.000, C 0.000 }
gfCNCPoint3[16751] = {X 51.7794, Y 71.1438, Z -4.6667, A 0.000, B 0.000, C 0.000 }
gfCNCPoint3[16752] = {X 49.6829, Y 71.3958, Z -4.6667, A 0.000, B 0.000, C 0.000 }
gfCNCPoint3[16753] = {X 47.5729, Y 71.4800, Z -4.6667, A 0.000, B 0.000, C 0.000 }
gfCNCPoint3[16754] = {X 40.6393, Y 71.4800, Z -4.6667, A 0.000, B 0.000, C 0.000 }
gfCNCPoint3[16755] = {X 38.8051, Y 71.4164, Z -4.6667, A 0.000, B 0.000, C 0.000 }
gfCNCPoint3[16756] = {X 36.9796, Y 71.2259, Z -4.6667, A 0.000, B 0.000, C 0.000 }
gfCNCPoint3[16757] = {X 34.3991, Y 72.0351, Z -4.6667, A 0.000, B 0.000, C 0.000 }
gfCNCPoint3[16758] = {X 31.7575, Y 72.6148, Z -4.6667, A 0.000, B 0.000, C 0.000 }
gfCNCPoint3[16759] = {X 30.3319, Y 73.1746, Z -4.6667, A 0.000, B 0.000, C 0.000 }
gfCNCPoint3[16760] = {X 28.8913, Y 73.6950, Z -4.6667, A 0.000, B 0.000, C 0.000 }
gfCNCPoint3[16761] = {X 108.0337, Y 73.6950, Z -4.6667, A 0.000, B 0.000, C 0.000 }
gfCNCPoint3[16762] = {X 110.0294, Y 72.3691, Z -4.6667, A 0.000, B 0.000, C 0.000 }
gfCNCPoint3[16763] = {X 112.1282, Y 71.2131, Z -4.6667, A 0.000, B 0.000, C 0.000 }
gfCNCPoint3[16764] = {X 113.1266, Y 70.7396, Z -4.6667, A 0.000, B 0.000, C 0.000 }
gfCNCPoint3[16765] = {X 114.1423, Y 70.3047, Z -4.6667, A 0.000, B 0.000, C 0.000 }
gfCNCPoint3[16766] = {X 117.4431, Y 66.6800, Z -4.6667, A 0.000, B 0.000, C 0.000 }
gfCNCPoint3[16767] = {X 111.9185, Y 66.6800, Z -4.6667, A 0.000, B 0.000, C 0.000 }
gfCNCPoint3[16768] = {X 111.5313, Y 66.6765, Z -4.6667, A 0.000, B 0.000, C 0.000 }
gfCNCPoint3[16769] = {X 111.1442, Y 66.6662, Z -4.6667, A 0.000, B 0.000, C 0.000 }
gfCNCPoint3[16770] = {X 111.2299, Y 64.2677, Z -4.6667, A 0.000, B 0.000, C 0.000 }
gfCNCPoint3[16771] = {X 109.1084, Y 64.0741, Z -4.6667, A 0.000, B 0.000, C 0.000 }
gfCNCPoint3[16772] = {X 107.0213, Y 63.6477, Z -4.6667, A 0.000, B 0.000, C 0.000 }
gfCNCPoint3[16773] = {X 105.0841, Y 64.0514, Z -4.6667, A 0.000, B 0.000, C 0.000 }
gfCNCPoint3[16774] = {X 103.1158, Y 64.2545, Z -4.6667, A 0.000, B 0.000, C 0.000 }
gfCNCPoint3[16775] = {X 101.1370, Y 64.2547, Z -4.6667, A 0.000, B 0.000, C 0.000 }
gfCNCPoint3[16776] = {X 99.1686, Y 64.0521, Z -4.6667, A 0.000, B 0.000, C 0.000 }
gfCNCPoint3[16777] = {X 97.2313, Y 63.6488, Z -4.6667, A 0.000, B 0.000, C 0.000 }
gfCNCPoint3[16778] = {X 95.6204, Y 63.9986, Z -4.6667, A 0.000, B 0.000, C 0.000 }
gfCNCPoint3[16779] = {X 93.9855, Y 64.2095, Z -4.6667, A 0.000, B 0.000, C 0.000 }
gfCNCPoint3[16780] = {X 92.3385, Y 64.2800, Z -4.6667, A 0.000, B 0.000, C 0.000 }
gfCNCPoint3[16781] = {X 85.8951, Y 64.2800, Z -4.6667, A 0.000, B 0.000, C 0.000 }
gfCNCPoint3[16782] = {X 85.5417, Y 64.2768, Z -4.6667, A 0.000, B 0.000, C 0.000 }
gfCNCPoint3[16783] = {X 85.1884, Y 64.2670, Z -4.6667, A 0.000, B 0.000, C 0.000 }
gfCNCPoint3[16784] = {X 83.3593, Y 65.5113, Z -4.6667, A 0.000, B 0.000, C 0.000 }
gfCNCPoint3[16785] = {X 81.4238, Y 66.5824, Z -4.6667, A 0.000, B 0.000, C 0.000 }
gfCNCPoint3[16786] = {X 79.3981, Y 67.4713, Z -4.6667, A 0.000, B 0.000, C 0.000 }
gfCNCPoint3[16787] = {X 77.2994, Y 68.1706, Z -4.6667, A 0.000, B 0.000, C 0.000 }
gfCNCPoint3[16788] = {X 75.1454, Y 68.6744, Z -4.6667, A 0.000, B 0.000, C 0.000 }
gfCNCPoint3[16789] = {X 72.9543, Y 68.9784, Z -4.6667, A 0.000, B 0.000, C 0.000 }
gfCNCPoint3[16790] = {X 70.7445, Y 69.0800, Z -4.6667, A 0.000, B 0.000, C 0.000 }
gfCNCPoint3[16791] = {X 64.1851, Y 69.0800, Z -4.6667, A 0.000, B 0.000, C 0.000 }
gfCNCPoint3[16792] = {X 62.0678, Y 68.9867, Z -4.6667, A 0.000, B 0.000, C 0.000 }
gfCNCPoint3[16793] = {X 59.9669, Y 68.7076, Z -4.6667, A 0.000, B 0.000, C 0.000 }
gfCNCPoint3[16794] = {X 57.8986, Y 68.2449, Z -4.6667, A 0.000, B 0.000, C 0.000 }
gfCNCPoint3[16795] = {X 55.8790, Y 67.6021, Z -4.6667, A 0.000, B 0.000, C 0.000 }
gfCNCPoint3[16796] = {X 53.8595, Y 68.2449, Z -4.6667, A 0.000, B 0.000, C 0.000 }
gfCNCPoint3[16797] = {X 51.7912, Y 68.7076, Z -4.6667, A 0.000, B 0.000, C 0.000 }
gfCNCPoint3[16798] = {X 49.6903, Y 68.9867, Z -4.6667, A 0.000, B 0.000, C 0.000 }
gfCNCPoint3[16799] = {X 47.5729, Y 69.0800, Z -4.6667, A 0.000, B 0.000, C 0.000 }
gfCNCPoint3[16800] = {X 40.6393, Y 69.0800, Z -4.6667, A 0.000, B 0.000, C 0.000 }
gfCNCPoint3[16801] = {X 38.6746, Y 68.9997, Z -4.6667, A 0.000, B 0.000, C 0.000 }
gfCNCPoint3[16802] = {X 36.7230, Y 68.7594, Z -4.6667, A 0.000, B 0.000, C 0.000 }
gfCNCPoint3[16803] = {X 34.8827, Y 69.3991, Z -4.6667, A 0.000, B 0.000, C 0.000 }
gfCNCPoint3[16804] = {X 33.0029, Y 69.9112, Z -4.6667, A 0.000, B 0.000, C 0.000 }
gfCNCPoint3[16805] = {X 31.0924, Y 70.2933, Z -4.6667, A 0.000, B 0.000, C 0.000 }
gfCNCPoint3[16806] = {X 29.6082, Y 70.8824, Z -4.6667, A 0.000, B 0.000, C 0.000 }
gfCNCPoint3[16807] = {X 28.1071, Y 71.4268, Z -4.6667, A 0.000, B 0.000, C 0.000 }
gfCNCPoint3[16808] = {X 27.6125, Y 71.5951, Z -4.6667, A 0.000, B 0.000, C 0.000 }
gfCNCPoint3[16809] = {X 27.1162, Y 71.7585, Z -4.6667, A 0.000, B 0.000, C 0.000 }
gfCNCPoint3[16810] = {X 25.5181, Y 72.2519, Z -4.6667, A 0.000, B 0.000, C 0.000 }
gfCNCPoint3[16811] = {X 23.9034, Y 72.6879, Z -4.6667, A 0.000, B 0.000, C 0.000 }
gfCNCPoint3[16812] = {X 23.9034, Y 76.0950, Z -4.6667, A 0.000, B 0.000, C 0.000 }
gfCNCPoint3[16813] = {X 108.8318, Y 76.0950, Z -4.6667, A 0.000, B 0.000, C 0.000 }
gfCNCPoint3[16814] = {X 110.4018, Y 74.9734, Z -4.6667, A 0.000, B 0.000, C 0.000 }
gfCNCPoint3[16815] = {X 112.0493, Y 73.9690, Z -4.6667, A 0.000, B 0.000, C 0.000 }
gfCNCPoint3[16816] = {X 113.7655, Y 73.0873, Z -4.6667, A 0.000, B 0.000, C 0.000 }
gfCNCPoint3[16817] = {X 115.5414, Y 72.3329, Z -4.6667, A 0.000, B 0.000, C 0.000 }
gfCNCPoint3[16818] = {X 123.7274, Y 63.3435, Z -4.6667, A 0.000, B 0.000, C 0.000 }
gfCNCPoint3[16819] = {X 121.7850, Y 63.8619, Z -4.6667, A 0.000, B 0.000, C 0.000 }
gfCNCPoint3[16820] = {X 119.7992, Y 64.1752, Z -4.6667, A 0.000, B 0.000, C 0.000 }
gfCNCPoint3[16821] = {X 117.7916, Y 64.2800, Z -4.6667, A 0.000, B 0.000, C 0.000 }
gfCNCPoint3[16822] = {X 111.9185, Y 64.2800, Z -4.6667, A 0.000, B 0.000, C 0.000 }
gfCNCPoint3[16823] = {X 111.5741, Y 64.2769, Z -4.6667, A 0.000, B 0.000, C 0.000 }
gfCNCPoint3[16824] = {X 111.2299, Y 64.2677, Z -4.6667, A 0.000, B 0.000, C 0.000 }
gfCNCPoint3[16825] = {X 111.3156, Y 61.8692, Z -4.6667, A 0.000, B 0.000, C 0.000 }
gfCNCPoint3[16826] = {X 109.8654, Y 61.7547, Z -4.6667, A 0.000, B 0.000, C 0.000 }
gfCNCPoint3[16827] = {X 108.4304, Y 61.5157, Z -4.6667, A 0.000, B 0.000, C 0.000 }
gfCNCPoint3[16828] = {X 107.0213, Y 61.1540, Z -4.6667, A 0.000, B 0.000, C 0.000 }
gfCNCPoint3[16829] = {X 105.0907, Y 61.6173, Z -4.6667, A 0.000, B 0.000, C 0.000 }
gfCNCPoint3[16830] = {X 103.1191, Y 61.8506, Z -4.6667, A 0.000, B 0.000, C 0.000 }
gfCNCPoint3[16831] = {X 101.1337, Y 61.8509, Z -4.6667, A 0.000, B 0.000, C 0.000 }
gfCNCPoint3[16832] = {X 99.1620, Y 61.6181, Z -4.6667, A 0.000, B 0.000, C 0.000 }
gfCNCPoint3[16833] = {X 97.2313, Y 61.1553, Z -4.6667, A 0.000, B 0.000, C 0.000 }
